(* CODESYS project fserror_0.2.0.1.library
   Company: FisoThemes
   DefaultNamespace: FsError
   Version: 0.2.0.1
   Placeholder: FsError
   Author: Goodwill Mzumala
   Description: A library that offers a set of functions for raising, handling, logging and querying error.
   Title: FsError

Project tree, tasks and I/O mapping:
  libraries: SysFile, * (System); SysTime, 3.5.9.0 (System); SysTypes2 Interfaces, * (System); Tc2_Standard, * (Beckhoff Automation GmbH); Tc2_System, * (Beckhoff Automation GmbH); Tc3_Module, * (Beckhoff Automation GmbH)
  DUTs/
    data type E_AdsReturnCode
    data type E_CodesysCmpError
    data type E_GeneralErrorCode
    data type T_DiskLoggerPath
    data type T_Error
    data type T_ErrorCode
    data type T_ErrorMessage
  GVLs/
    global variables GVL_ErrorDescriptors
  ITFs/
    interface I_Error: Code, Descriptor, IsNotRaised, IsRaised, LogMessage, Message, Timestamp
    interface I_ErrorDescriptor: GetDescription
    interface I_ErrorLogger: Invoke
    interface I_ErrorTimestamp: AsDateTime, GetDate, GetTimeOfDay, Raw
    interface I_MutableError: CopyFrom, RaiseError, SetDescriptor, SetTimestamp
  PARAMs/
    global variables PARAM_Constants
  POUs/
    Error Descriptors/
      function block FB_AdsReturnCodesDescriptor [ST]: GetDescription
      function block FB_CodesysCmpErrorDescriptor [ST]: GetDescription
      function block FB_GeneralCodesDescriptor [ST]: GetDescription
    Errors/
      function F_CreateError [ST]
      function F_CreateErrorFromStartRange [ST]
      function block FB_Error [ST]: Code, Descriptor, IsNotRaised, IsRaised, LogMessage, Message, Timestamp
      function block FB_MutableError [ST]: CopyFrom, RaiseError, SetDescriptor, SetTimestamp
    Loggers/
      function block FB_AdsErrorLogger [ST]: Invoke, SetMessageType
      function block FB_DiskErrorLogger [ST]: CreateLogEntry, AutoFlush, Close, Delimiter, FB_exit, FB_init, Flush, Invoke, IsOpen, LineEnding, Open, SetDelimiter, SetLineEnding, SetTextQualifier, TextQualifier
    Timestamp/
      function block FB_ErrorTimestamp [ST]: AsDateTime, GetDate, GetTimeOfDay, Raw
    program PLAYGROUND [ST]
  Project Information/
    function F_GetCompany [ST]
    function F_GetTitle [ST]
    function F_GetVersion [ST]
  UML/
    Error Class Diagram
    Error Descriptor Class Diagram
    Error Logger Class Diagram
    Error Timestamp Class Diagram
  Version/
    global variables Global_Version
*)

// DUTs/E_AdsReturnCode
// All ADS error codes.
// Source: https://github.com/Roald87/TcError/blob/main/TcError/TcError/ADS/AdsErrorCodes.TcDUT
// See end for licensing information.
{attribute 'qualified_only'}
{attribute 'to_string'}
TYPE E_AdsReturnCode :
(
    ERR_NOERROR 					:= 0,					// No error.
    ERR_INTERNAL,  											// Internal error.
    ERR_NORTIME,  											// No real-time.
    ERR_ALLOCLOCKEDMEM,  									// Allocation locked – memory error.
    ERR_INSERTMAILBOX,  									// Mailbox full – the ADS message could not be sent. Reducing the number of ADS messages per cycle will help.
    ERR_WRONGRECEIVEHMSG,  									// Wrong HMSG.
    ERR_TARGETPORTNOTFOUND,  								// Target port not found – ADS server is not started or is not reachable.
    ERR_TARGETMACHINENOTFOUND,  							// Target computer not found – AMS route was not found.
    ERR_UNKNOWNCMDID, 										// Unknown command ID.
    ERR_BADTASKID,  										// Invalid task ID.
    ERR_NOIO,  												// No IO.
	ERR_UNKNOWNAMSCMD,  									// Unknown AMS command.
    ERR_WIN32ERROR,  										// Win32 error.
    ERR_PORTNOTCONNECTED,  									// Port not connected.
    ERR_INVALIDAMSLENGTH,  									// Invalid AMS length.
    ERR_INVALIDAMSNETID,  									// Invalid AMS Net ID.
    ERR_LOWINSTLEVEL,  										// Installation level is too low –TwinCAT 2 license error.
    ERR_NODEBUGINTAVAILABLE,  								// No debugging available.
    ERR_PORTDISABLED,  										// Port disabled – TwinCAT system service not started.
    ERR_PORTALREADYCONNECTED,  								// Port already connected.
	ERR_AMSSYNC_W32ERROR,  									// AMS Sync Win32 error.
	ERR_AMSSYNC_TIMEOUT,  									// AMS Sync Timeout.
    ERR_AMSSYNC_AMSERROR,  									// AMS Sync error.
    ERR_AMSSYNC_NOINDEXINMAP,  								// No index map for AMS Sync available.
    ERR_INVALIDAMSPORT,  									// Invalid AMS port.
    ERR_NOMEMORY,  											// No memory.
    ERR_TCPSEND,  											// TCP send error.
    ERR_HOSTUNREACHABLE,  									// Host unreachable.
    ERR_INVALIDAMSFRAGMENT,  								// Invalid AMS fragment.
    ERR_TLSSEND,  											// TLS send error – secure ADS connection failed.
    ERR_ACCESSDENIED,  										// Access denied – secure ADS access denied.
    ROUTERERR_NOLOCKEDMEMORY 				:= 1280,		// Locked memory cannot be allocated.
    ROUTERERR_RESIZEMEMORY,  								// The router memory size could not be changed.
	ROUTERERR_MAILBOXFULL,  								// The mailbox has reached the maximum number of possible messages.
    ROUTERERR_DEBUGBOXFULL,  								// The Debug mailbox has reached the maximum number of possible messages.
    ROUTERERR_UNKNOWNPORTTYPE,  							// The port type is unknown.
    ROUTERERR_NOTINITIALIZED,  								// The router is not initialized.
    ROUTERERR_PORTALREADYINUSE,  							// The port number is already assigned.
    ROUTERERR_NOTREGISTERED,  								// The port is not registered.
    ROUTERERR_NOMOREQUEUES,  								// The maximum number of ports has been reached.
    ROUTERERR_INVALIDPORT,  								// The port is invalid.
    ROUTERERR_NOTACTIVATED,  								// The router is not active.
    ROUTERERR_FRAGMENTBOXFULL,  							// The mailbox has reached the maximum number for fragmented messages.
    ROUTERERR_FRAGMENTTIMEOUT,  							// A fragment timeout has occurred.
	ROUTERERR_TOBEREMOVED,  								// The port is removed.
    ADSERR_DEVICE_ERROR 					:= 1792,  		// General device error.
    ADSERR_DEVICE_SRVNOTSUPP,  								// Service is not supported by the server.
    ADSERR_DEVICE_INVALIDGRP,  								// Invalid index group.
    ADSERR_DEVICE_INVALIDOFFSET,  							// Invalid index offset.
    ADSERR_DEVICE_INVALIDACCESS,  							// Reading or writing not permitted.
    ADSERR_DEVICE_INVALIDSIZE,  							// Parameter size not correct.
    ADSERR_DEVICE_INVALIDDATA,  							// Invalid data values.
    ADSERR_DEVICE_NOTREADY,  								// Device is not ready to operate.
    ADSERR_DEVICE_BUSY,  									// Device is busy.
    ADSERR_DEVICE_INVALIDCONTEXT,  							// Invalid operating system context. This can result from use of ADS function blocks in different tasks. It may be possible to resolve this through Multi-task data access synchronization in the PLC.
    ADSERR_DEVICE_NOMEMORY,  								// Insufficient memory.
    ADSERR_DEVICE_INVALIDPARM,  							// Invalid parameter values.
    ADSERR_DEVICE_NOTFOUND,  								// Not found (files, ...).
	ADSERR_DEVICE_SYNTAX,  									// Syntax error in file or command.
    ADSERR_DEVICE_INCOMPATIBLE,  							// Objects do not match.
    ADSERR_DEVICE_EXISTS,  									// Object already exists.
    ADSERR_DEVICE_SYMBOLNOTFOUND,  							// Symbol not found.
    ADSERR_DEVICE_SYMBOLVERSIONINVALID,  					// Invalid symbol version. This can occur due to an online change. Create a new handle.
    ADSERR_DEVICE_INVALIDSTATE,  							// Device (server) is in invalid state.
    ADSERR_DEVICE_TRANSMODENOTSUPP,  						// AdsTransMode not supported.
    ADSERR_DEVICE_NOTIFYHNDINVALID,  						// Notification handle is invalid.
    ADSERR_DEVICE_CLIENTUNKNOWN,  							// Notification client not registered.
    ADSERR_DEVICE_NOMOREHDLS,  								// No further handle available.
    ADSERR_DEVICE_INVALIDWATCHSIZE,  						// Notification size too large.
    ADSERR_DEVICE_NOTINIT,  								// Device not initialized.
    ADSERR_DEVICE_TIMEOUT,  								// Device has a timeout.
    ADSERR_DEVICE_NOINTERFACE,  							// Interface query failed.
    ADSERR_DEVICE_INVALIDINTERFACE,  						// Wrong interface requested.
    ADSERR_DEVICE_INVALIDCLSID,  							// Class ID is invalid.
    ADSERR_DEVICE_INVALIDOBJID,  							// Object ID is invalid.
    ADSERR_DEVICE_PENDING,  								// Request pending.
    ADSERR_DEVICE_ABORTED,  								// Request is aborted.
    ADSERR_DEVICE_WARNING,  								// Signal warning.
    ADSERR_DEVICE_INVALIDARRAYIDX,  						// Invalid array index.
    ADSERR_DEVICE_SYMBOLNOTACTIVE,  						// Symbol not active.
    ADSERR_DEVICE_ACCESSDENIED,  							// Access denied.
    ADSERR_DEVICE_LICENSENOTFOUND,  						// Missing license.
    ADSERR_DEVICE_LICENSEEXPIRED,  							// License expired.
    ADSERR_DEVICE_LICENSEEXCEEDED,  						// License exceeded.
    ADSERR_DEVICE_LICENSEINVALID,  							// Invalid license.
    ADSERR_DEVICE_LICENSESYSTEMID,  						// License problem: System ID is invalid.
    ADSERR_DEVICE_LICENSENOTIMELIMIT,  						// License not limited in time.
    ADSERR_DEVICE_LICENSEFUTUREISSUE,  						// License problem: Time in the future.
    ADSERR_DEVICE_LICENSETIMETOLONG,  						// License period too long.
    ADSERR_DEVICE_EXCEPTION,  								// Exception at system startup.
	ADSERR_DEVICE_LICENSEDUPLICATED,  						// License file read twice.
	ADSERR_DEVICE_SIGNATUREINVALID, 						// License file read twice.
	ADSERR_DEVICE_CERTIFICATEINVALID,  						// Invalid certificate.
    ADSERR_DEVICE_LICENSEOEMNOTFOUND,  						// Public key not known from OEM.
    ADSERR_DEVICE_LICENSERESTRICTED,  						// License not valid for this system ID.
    ADSERR_DEVICE_LICENSEDEMODENIED,  						// Demo license prohibited.
    ADSERR_DEVICE_INVALIDFNCID,  							// Invalid function ID.
    ADSERR_DEVICE_OUTOFRANGE,  								// Outside the valid range.
    ADSERR_DEVICE_INVALIDALIGNMENT,  						// Invalid alignment.
    ADSERR_DEVICE_LICENSEPLATFORM,  						// Invalid platform level.
    ADSERR_DEVICE_FORWARD_PL,  								// Context – forward to passive level.
    ADSERR_DEVICE_FORWARD_DL,  								// Context – forward to dispatch level.
    ADSERR_DEVICE_FORWARD_RT,  								// Context – forward to real-time.
    ADSERR_CLIENT_ERROR 					:= 1856,  		// Client error.
    ADSERR_CLIENT_INVALIDPARM,  							// Service contains an invalid parameter.
    ADSERR_CLIENT_LISTEMPTY,  								// Polling list is empty.
    ADSERR_CLIENT_VARUSED,  								// Var connection already in use.
    ADSERR_CLIENT_DUPLINVOKEID,  							// The called ID is already in use.
    ADSERR_CLIENT_SYNCTIMEOUT,  							// Timeout has occurred – the remote terminal is not responding in the specified ADS timeout. The route setting of the remote terminal may be configured incorrectly.
    ADSERR_CLIENT_W32ERROR,  								// Error in Win32 subsystem.
    ADSERR_CLIENT_TIMEOUTINVALID,  							// Invalid client timeout value.
    ADSERR_CLIENT_PORTNOTOPEN,  							// Port not open.
    ADSERR_CLIENT_NOAMSADDR,  								// No AMS address.
    ADSERR_CLIENT_SYNCINTERNAL,  							// Internal error in Ads sync.
	ADSERR_CLIENT_ADDHASH,  								// Hash table overflow.
    ADSERR_CLIENT_REMOVEHASH,  								// Key not found in the table.
    ADSERR_CLIENT_NOMORESYM,  								// No symbols in the cache.
    ADSERR_CLIENT_SYNCRESINVALID,  							// Invalid response received.
    ADSERR_CLIENT_SYNCPORTLOCKED,  							// Sync Port is locked.
    RTERR_INTERNAL 							:= 4096,  		// Internal error in the real-time system.
    RTERR_BADTIMERPERIODS,  								// Timer value is not valid.
    RTERR_INVALIDTASKPTR,  									// Task pointer has the invalid value 0 (zero).
    RTERR_INVALIDSTACKPTR,  								// Stack pointer has the invalid value 0 (zero).
    RTERR_PRIOEXISTS,  										// The request task priority is already assigned.
    RTERR_NOMORETCB,  										// No free TCB (Task Control Block) available. The maximum number of TCBs is 64.
    RTERR_NOMORESEMAS,  									// No free semaphores available. The maximum number of semaphores is 64.
    RTERR_NOMOREQUEUES,  									// No free space available in the queue. The maximum number of positions in the queue is 64.
    RTERR_EXTIRQALREADYDEF					:= 4109,  		// An external synchronization interrupt is already applied.
    RTERR_EXTIRQNOTDEF,  									// No external sync interrupt applied.
    RTERR_EXTIRQINSTALLFAILED,  							// Application of the external synchronization interrupt has failed.
    RTERR_IRQLNOTLESSOREQUAL,  								// Call of a service function in the wrong context
    RTERR_VMXNOTSUPPORTED					:= 4119,  		// Intel VT-x extension is not supported.
    RTERR_VMXDISABLED,  									// Intel VT-x extension is not enabled in the BIOS.
    RTERR_VMXCONTROLSMISSING,  								// Missing function in Intel VT-x extension.
    RTERR_VMXENABLEFAILS,  									// Activation of Intel VT-x fails.
	WSAETIMEDOUT							:= 10060,		// A connection timeout has occurred while establishing the connection. Either the remote terminal did not respond properly after a certain period of time, or the established connection could not be maintained because the connected host did not respond.
    WSAECONNREFUSED							:= 10061,		// Connection refused. Connection couldn't be established because the target computer has rejected it. Error can result from an attempt to connect to a service that is inactive on the external host, i.e. a service for which no server application is running.
    WSAEHOSTUNREACH							:= 10065,		// No route to host - a socket operation referred to an unavailable host.
	ERR_UNKNOWN                       		:= 4294967294	// Unknown ADS error code.
)LINT;
END_TYPE
(*
	MIT License
	
	Copyright (c) 2022 Roald87
	
	Permission is hereby granted, free of charge, to any person obtaining a copy
	of this software and associated documentation files (the "Software"), to deal
	in the Software without restriction, including without limitation the rights
	to use, copy, modify, merge, publish, distribute, sublicense, and/or sell
	copies of the Software, and to permit persons to whom the Software is
	furnished to do so, subject to the following conditions:
	
	The above copyright notice and this permission notice shall be included in all
	copies or substantial portions of the Software.
	
	THE SOFTWARE IS PROVIDED "AS IS", WITHOUT WARRANTY OF ANY KIND, EXPRESS OR
	IMPLIED, INCLUDING BUT NOT LIMITED TO THE WARRANTIES OF MERCHANTABILITY,
	FITNESS FOR A PARTICULAR PURPOSE AND NONINFRINGEMENT. IN NO EVENT SHALL THE
	AUTHORS OR COPYRIGHT HOLDERS BE LIABLE FOR ANY CLAIM, DAMAGES OR OTHER
	LIABILITY, WHETHER IN AN ACTION OF CONTRACT, TORT OR OTHERWISE, ARISING FROM,
	OUT OF OR IN CONNECTION WITH THE SOFTWARE OR THE USE OR OTHER DEALINGS IN THE
	SOFTWARE.
*)

// DUTs/E_CodesysCmpError
 // Error codes are found @ CmpErrors.Errors.<variable> from the CmpErrors2 Interfaces library.
 // See: https://help.codesys.com/webapp/Errors;product=CmpErrors2_Itfs;version=3.5.15.0
{attribute 'qualified_only'}
{attribute 'to_string'}
TYPE E_CodesysCmpError :
(
	ERR_OK 						 := 16#0,	//	Ok
	ERR_FAILED 					 := 16#1, 	//	General error - To be used only for internal errors
	ERR_PARAMETER 				 := 16#2, 	//	Invalid parameter for this operation
	ERR_NOT_INITIALIZED 		 := 16#3, 	//	Function cannot be executed, since component has not been initialized yet. It may work later, though
	ERR_VERSION 				 := 16#4, 	//	Version conflict
	ERR_TIMEOUT 				 := 16#5, 	//	Operation timed out
	ERR_NO_BUFFER 				 := 16#6, 	//	Insufficient memory to carry out the request
	ERR_PENDING 				 := 16#A, 	//	For async-calls: call not complete, yet
	ERR_NUM_PENDING 			 := 16#B, 	//  Too many pending calls. Try later
	ERR_NOT_IMPLEMENTED 		 := 16#C, 	//  The function is not implemented
	ERR_INVALID_ID 				 := 16#D, 	//  No object with the provided id found
	ERR_OVERFLOW 				 := 16#E, 	//	Integer overflow
	ERR_BUFFER_SIZE 			 := 16#F, 	//	The size of a buffer is too small OR invalid
	ERR_NO_OBJECT 				 := 16#10,	//	No object with this specified name available
	ERR_NO_MEMORY 				 := 16#11,	//  No heap memory available
	ERR_DUPLICATE 				 := 16#12, 	//  An object with the same name is still available
	ERR_MEMORY_OVERWRITE 		 := 16#13,  //  Heap memory was written out of bounds! Memory overwrite error
	ERR_INVALID_HANDLE 			 := 16#14,  //  Invalid handle to an object
	ERR_END_OF_0BJECT 			 := 16#15,  //  End OF object reached
	ERR_NO_CHANGE 				 := 16#16,  //  No changes done
	ERR_INVALID_INTERFACE 		 := 16#17,  //  Invalid or unknown interface
	ERR_NOT_SUPPORTED 			 := 16#18,  //  Functionality not supported
	ERR_NO_ACCESS_RIGHTS 		 := 16#19,  //  No access rights for this operation
	ERR_OUT_OF_LIMITS 			 := 16#1A,  //  Specified limits of a resource exceeded
	ERR_ENTRIES_REMAINING 		 := 16#1B,  //  Remaining entries that could not be transmitted because of buffer limitation
	ERR_INVALID_SESSION_ID 		 := 16#1C,  //  Invalid online sessionid
	ERR_EXCEPTION 				 := 16#1D,  //  Exception occurred
	ERR_SIGNATURE_MISMATCH 		 := 16#1E,	//	Signature mismatch of an api function
	ERR_VERSION_MISMATCH 		 := 16#1F,	//	Version mismatch
	ERR_TYPE_MISMATCH 			 := 16#20,	//	Type mismatch
	ERR_ID_MISMATCH 			 := 16#21,	//	ID mismatch
	ERR_NO_CONSISTENCY 			 := 16#22,	//	Consistency error
	ERR_NO_COMM_CYCLE 			 := 16#23,	//	No COMM_CYCLE needed
	ERR_DONT_SUSPEND_TASK 		 := 16#24,	//	Do not suspend task after an exception
	ERR_MEMORY_LOCK_FAILED 		 := 16#25,	//	Memory cannot be locked in this operation
	ERR_LICENSE_MISSING 		 := 16#26,	//	License missing for the runtime
	ERR_OPERATION_DENIED 		 := 16#27,	//	Operation denied 
	ERR_DEVICE 					 := 16#28,	//	Device error
	ERR_DISK_FULL 				 := 16#29,	//	Disk full
	ERR_CRC_FAILED 				 := 16#30,	//	Internal use in runtime
	ERR_MEDIA_ERASE 			 := 16#31,	//	Internal use in runtime
	ERR_FILE_ERROR 				 := 16#32,	//	File error. e.g. cannot open a file for writing because it could be write protected
	ERR_NO_RETAIN_MEMORY 		 := 16#33,	//	No retain memory available
	ERR_OUT_OF_LIMITS_MIN 		 := 16#34,	//	Specified minimum-limit of a resource exceeded
	ERR_OUT_OF_LIMITS_MAX 		 := 16#35,	//	Specified maximum-limit of a resource exceeded
	ERR_SIZE_MISMATCH 			 := 16#36,	//	Size mismatch
	ERR_CALL_AGAIN 				 := 16#37,	//	Operation is not yet finished, call function again to proceed
	ERR_NOTHING_TO_DO 			 := 16#38,	//	Operation has nothing to do. No execution.
	ERR_SECURITY_CHECKS_FAILED 	 := 16#39,	//	Some security checks have failed. /* This is a generic error code to report this error over public channels. In this case the error code doesn’t provide a detailed cause for the error. */
	ERR_INVALID_SEQUENCE 		 := 16#3A,	//	 
	ERR_INVALID_REFERENCE 		 := 16#3B,	//	Dereferencing an IEC reference in IecVarAccess failed due to invalid destination address, e. G. NULL.
	ERR_CONVERSION_INCOMPLETE 	 := 16#3C,	//	Conversion of string encodings was not lossless.
	ERR_SOCK_NOT_INITIALIZED 	 := 16#201, //  Socket errors (range: 0x0200 - 0X02FF)
	ERR_SOCK_NOT_SOCKET 		 := 16#202, //  The provided socket handle is invalid
	ERR_SOCK_AF_UNSUPPORTED 	 := 16#203, //  The address family is not supported
	ERR_SOCK_PROTO_UNSUPPORTED   := 16#204, //  Protocol is not supported 
	ERR_SOCK_NO_BUFFER 			 := 16#205, //  Not enough buffer to handle the request 
	ERR_SOCK_WOULD_BLOCK 		 := 167206, //  Socket is in nonblocking mode but this call would block 
	ERR_SOCK_ADDR_INUSE 		 := 16#207, //  The provided address is already in use 
	ERR_SOCK_ADDR_NOT_AVAILABLE  := 16#208, //  The provided address is not available on THIS computer 
	ERR_SOCK_CONN_REFUSED 		 := 16#209, //  Connection has been refused by the remote host 
	ERR_SOCK_TIMEDOUT 			 := 16#20A, //  Operation timed out
	ERR_SOCK_HOST_NOT_FOUND 	 := 16#20B, //  The host has NOT been found
	ERR_SOCK_HOST_UNREACHABLE  	 := 16#20C, //  Host is unreachable
	ERR_SOCK_1S_CONNECTED 		 := 16#20D, //  Socket is already connected
	ERR_SOCK_NOT_CONNECTED 		 := 16#20E, //  The socket is not connected
	ERR_SOCK_SHUTDOWN 			 := 16#20F, //  Shutdown has been called on the socket 
	ERR_SOCK_MSGSIZE 			 := 16#210, //  For sockets of type DGRAM. The package to send exceeds the maximum package size 
	ERR_SOCK_CLOSED 			 := 16#211, //  Socket has been gracefully closed. No more send/receives allowed 
	ERR_L7_TAG_MISSING 			 := 16#300,	//  Tag missing in online communication buffer
	ERR_L7_UNKNOWN_CMD_GROUP 	 := 16#301,	//  Unknown command group
	ERR_L7_UNKNOWN_CMD 			 := 16#302,	//  Unknown command (within a valid command group)
	ERR_L7_INCOMPLETE 			 := 16#303	//  Level 7 service incomplete
)LINT;
END_TYPE

// DUTs/E_GeneralErrorCode
// List of general error codes used in a system.
{attribute 'qualified_only'}
{attribute 'to_string'}
TYPE E_GeneralErrorCode :
(
	{region "General Errors (1-99)"}
	ERR_NO_ERROR                    := 0,      // No error.
	ERR_GENERAL_ERROR               := 1,      // General error - To be used only for internal errors
	ERR_INVALID_PARAMETER           := 2,      // Invalid parameter for this operation
	ERR_NOT_INITIALIZED             := 3,      // Function cannot be executed since the component has not been initialized yet. It may work later, though
	ERR_VERSION_CONFLICT            := 4,      // Version conflict
	{endregion}
	
	{region "Overflow Errors (100-119)"}
	ERR_INTEGER_OVERFLOW            := 100,    // Integer overflow
	ERR_BUFFER_OVERFLOW             := 101,    // Buffer overflow
	ERR_STACK_OVERFLOW              := 102,    // Stack overflow
	ERR_HEAP_OVERFLOW               := 103,    // Heap overflow
	{endregion}
	
	{region "Buffer Errors (120-139)"}
	ERR_NO_BUFFER                   := 120,    // No buffer available
	ERR_BUFFER_UNDERFLOW            := 121,    // Buffer underflow
	ERR_BUFFER_FULL                 := 123,    // Buffer is full
	{endregion}
	
	{region "Configuration and Settings Errors (140-159)"}
	ERR_INVALID_CONFIGURATION       := 140,    // Invalid configuration or settings
	ERR_CONFIGURATION_MISSING       := 141,    // Required configuration setting or parameter is missing
	{endregion}
	
	{region "Network Errors (200-249)"}
	ERR_NETWORK_ERROR               := 200,    // Network communication or connectivity issues
	ERR_TIMEOUT_CONNECT             := 201,    // Connection timeout
	ERR_TIMEOUT_READ                := 202,    // Read timeout
	ERR_TIMEOUT_WRITE               := 203,    // Write timeout
	ERR_UNSUPPORTED_FORMAT          := 204,    // Unsupported data format
	ERR_TOO_MANY_REQUESTS           := 205,    // Too many requests or actions in a short period
	{endregion}
	
	{region "Stream Errors (250-299)"}
	ERR_STREAM_ERROR                := 250,    // Generic stream error
	ERR_STREAM_NOT_FOUND            := 251,    // Stream not found
	ERR_STREAM_READ_FAILED          := 252,    // Stream read operation failed
	ERR_STREAM_WRITE_FAILED         := 253,    // Stream write operation failed
	ERR_STREAM_PERMISSION_DENIED    := 254,    // Stream operation permission denied
	ERR_STREAM_ALREADY_EXISTS       := 255,    // Stream already exists
	{endregion}
	
	{region "Resource Errors (300-339)"}
	ERR_NOT_FOUND                   := 300,    // The resource has not been found
	ERR_PERMISSION_DENIED           := 301,    // Permission denied
	ERR_DATA_NOT_AVAILABLE          := 302,    // Requested data is not available
	ERR_OUT_OF_BOUNDS               := 303,    // Value is outside the valid range
	ERR_DATA_CORRUPTED              := 304,    // Data corruption or integrity issues
	ERR_INVALID_INTERFACE           := 305,    // Invalid or unknown interface
	ERR_INVALID_REFERENCE           := 306,    // Dereferencing an IEC reference in IecVarAccess failed due to an invalid destination address, e.g., NULL.
	ERR_INVALID_POINTER             := 307,    // Invalid pointer
	ERR_INVALID_HANDLE              := 308,    // Invalid handle to an object
	ERR_MIN_LIMIT_EXCEEDED          := 309,    // Specified minimum-limit of the resource exceeded
	ERR_MAX_LIMIT_EXCEEDED          := 310,    // Specified maximum-limit of the resource exceeded
	ERR_DUPLICATE                   := 311,    // The resource already exists
	{endregion}
	
	{region "Hardware Errors (400-449)"}
	ERR_HARDWARE_FAILURE            := 400,    // Hardware malfunctions or failures
	{endregion}
	
	{region "Resource Management Errors (500-549)"}
	ERR_RESOURCE_BUSY               := 500,    // Resource is currently in use and cannot be accessed
	ERR_RESOURCE_LOCKED             := 501,    // Resource is locked and cannot be accessed
	{endregion}
	
	{region "State and Operation Errors (600-649)"}
	ERR_INVALID_STATE               := 600,    // Invalid state for the requested operation
	ERR_INVALID_OPERATION           := 601,    // Requested operation is not allowed or valid in the current context
	ERR_OPERATION_TIMEOUT           := 602,    // Operation timed out
	ERR_OPERATION_FAILED            := 603,    // Operation failed
	{endregion}
	
	{region "Service and API Errors (700-749)"}
	ERR_EXTERNAL_SERVICE_FAILURE    := 700,    // Failure in an external service or API
	ERR_UNAVAILABLE_SERVICE         := 701,    // Required service or component is not available
	{endregion}
	
	{region "Data Conversion Errors (800-849)"}
	ERR_INVALID_INPUT               := 800,   // Invalid or unexpected input provided
	ERR_INVALID_CONVERSION          := 801,   // Invalid data conversion
	ERR_INVALID_COMPARISON          := 802,   // Invalid comparison
	ERR_TYPE_MISMATCH               := 803,   // Type mismatch
	ERR_SIZE_MISMATCH               := 804,   // Size mismatch
	{endregion}
	
	{region "Security Errors (900-949)"}
	ERR_SECURITY_CHECKS_FAILED      := 900,   // Some security checks have failed. (Generic error for reporting over public channels)
	ERR_AUTHENTICATION_FAILED       := 901,   // Authentication process failed
	ERR_AUTHORIZATION_FAILED        := 902,   // Authorization failed due to insufficient permissions
	{endregion}
	
	{region "Memory Errors (1000-1049)"}
	ERR_MEMORY_ALLOCATION_FAILED    := 1000,  // Memory allocation failed
	ERR_INSUFFICIENT_MEMORY         := 1001,  // Insufficient memory to carry out the request
	ERR_INSUFFICIENT_MEMORY_FULL    := 1002,  // Memory full
	{endregion}
	
	{region "File Errors (1100-1149)"}
	ERR_FILE_NOT_FOUND              := 1100,  // The specified file was not found
	ERR_FILE_READ_FAILED            := 1101,  // File read operation failed
	ERR_FILE_WRITE_FAILED           := 1102,  // File write operation failed
	ERR_FILE_PERMISSION_DENIED      := 1103,  // File operation permission denied
	ERR_FILE_ALREADY_EXISTS         := 1104,  // File already exists
	ERR_FILE_TOO_LARGE              := 1105,  // File size exceeds the maximum allowed size
	ERR_FILE_FORMAT_UNSUPPORTED     := 1106,  // Unsupported file format
	ERR_FILE_NOT_OPEN				:= 1107,  // File isn't open
	ERR_FILE_INVALID_HANDLE			:= 1108,  // File handle is invalid
	{endregion}
	
	{region "Directory Errors (1150-1199)"}
	ERR_DIRECTORY_NOT_FOUND         := 1150,  // The specified directory was not found
	ERR_DIRECTORY_READ_FAILED       := 1151,  // Directory read operation failed
	ERR_DIRECTORY_WRITE_FAILED      := 1152,  // Directory write operation failed
	ERR_DIRECTORY_PERMISSION_DENIED := 1153,  // Directory operation permission denied
	ERR_DIRECTORY_NOT_EMPTY         := 1154,  // Directory is not empty
	ERR_DIRECTORY_ALREADY_EXISTS    := 1155,  // Directory already exists
	ERR_DIRECTORY_NOT_OPEN			:= 1157,  // Directory isn't open
	ERR_DIRECTORY_INVALID_HANDLE	:= 1158,  // Directory handle is invalid
	{endregion}
	
	{region "Cache Errors (1200-1249)"}
	ERR_CACHE_MISS                  := 1200,  // Cache miss occurred
	ERR_CACHE_WRITE_FAILED          := 1201,  // Cache write operation failed
	{endregion}
	
	{region "Serialization/Deserialization Errors (1300-1349)"}
	ERR_SERIALIZATION_FAILED        := 1300,  // Data serialization failed
	ERR_DESERIALIZATION_FAILED      := 1301,  // Data deserialization failed
	{endregion}
	
	{region "Threading and Concurrency Errors (1400-1449)"}
	ERR_THREAD_CREATION_FAILED      := 1400,  // Thread creation failed
	ERR_DEADLOCK_DETECTED           := 1401,  // Deadlock detected
	ERR_CONCURRENCY_VIOLATION       := 1402,  // Concurrency violation
	{endregion}
	
	{region "Protocol Errors (1500-1549)"}
	ERR_PROTOCOL_VIOLATION          := 1500,  // Protocol violation detected
	ERR_UNSUPPORTED_PROTOCOL        := 1501,  // Unsupported protocol
	{endregion}
	
	{region "User Errors (1600-1699)"}
	ERR_USER_INPUT_INVALID          := 1600,  // User input is invalid or malformed
	ERR_USER_INPUT_TOO_LONG         := 1601,  // User input exceeds maximum allowed length
	ERR_USER_INPUT_TOO_SHORT        := 1602,  // User input is shorter than the minimum required length
	ERR_USER_AUTHENTICATION_FAILED  := 1603,  // User authentication failed
	ERR_USER_AUTHORIZATION_FAILED   := 1604,  // User is not authorized to perform this action
	ERR_USER_ACCOUNT_LOCKED         := 1605,  // User account is locked
	ERR_USER_ACCOUNT_DISABLED       := 1606,  // User account is disabled
	ERR_USER_SESSION_EXPIRED        := 1607,  // User session has expired
	ERR_USER_ALREADY_EXISTS         := 1608,  // User already exists
	ERR_USER_NOT_FOUND              := 1609,  // User not found
	ERR_USER_CANCELLED              := 1610,  // User cancelled the operation or action
	{endregion}
	
	{region "Internal additional errors (5000-5099)"}
	ERR_NOTHING_TO_DO               := 5000,  // Operation has nothing to do. No execution.
	ERR_FUNCTION_NOT_SUPPORTED      := 5001,  // Functionality not supported
	{endregion}
	
	{region "Custom errors (10000-99999)"}
	ERR_CUSTOM_ERROR_BEGIN          := 10_000,  // Custom or application-specific error codes can be defined starting from here
	ERR_CUSTOM_ERROR_END          	:= 99_999,  // Custom or application-specific error codes definition ends here
	{endregion}
	
	{region "Codesys errors (200000-299999)"} 
	ERR_CODESYS_BEGIN				:= 100_000, // Start range of Codesys errors in the context of general errors
	ERR_CODESYS_END					:= 999_999,	// End range of Codesys errors in the context of general errors
	{endregion}
	
	{region "ADS errors (1,000,000,000-...)"} 
	ERR_ADS_RETURN_CODE_BEGIN		:= 1_000_000_000, // Start range of ADS return codes in the context of general errors
	ERR_ADS_RETURN_CODE_END 		:= ERR_ADS_RETURN_CODE_BEGIN + 4_294_967_294 // End range of ADS return codes in the context of general errors
	{endregion}
) LINT;
END_TYPE

// DUTs/T_DiskLoggerPath
TYPE T_DiskLoggerPath : STRING(PARAM_Constants.DISK_LOGGER_PATH_LENGTH); END_TYPE

// DUTs/T_Error
// Alias for the error object.
TYPE T_Error : FB_Error; END_TYPE

// DUTs/T_ErrorCode
// Alias for error code.
TYPE T_ErrorCode : LINT; END_TYPE

// DUTs/T_ErrorMessage
// Alias for error messages as strings with a predefined maximum length.
// Length of message can be changed in the **Library_Parameters**.
TYPE T_ErrorMessage : STRING(PARAM_Constants.ERROR_MESSAGE_SIZE); END_TYPE

// GVLs/GVL_ErrorDescriptors
{attribute 'qualified_only'}
VAR_GLOBAL
	fbAdsReturnCodes	: FB_AdsReturnCodesDescriptor;
	fbCodesysCmpErrors 	: FB_CodesysCmpErrorDescriptor;
	fbGeneralErrorCodes	: FB_GeneralCodesDescriptor;
END_VAR

// PARAMs/PARAM_Constants
// Main parameters for the library.
{attribute 'qualified_only'}
VAR_GLOBAL CONSTANT
	ERROR_MESSAGE_SIZE 				: __UXINT := 255; // String length of an error message.
	DISK_LOGGER_PATH_LENGTH			: __UXINT := 300; // String length of disk logger path.
END_VAR

// Version/Global_Version
{attribute 'TcGenerated'}
{attribute 'no-analysis'}
{attribute 'linkalways'}
// This function has been automatically generated from the project information.
VAR_GLOBAL CONSTANT
	{attribute 'const_non_replaced'}
	stLibVersion_FsError : ST_LibVersion := (iMajor := 0, iMinor := 2, iBuild := 0, iRevision := 1, nFlags := 0, sVersion := '0.2.0.1');
END_VAR

// ITFs/I_Error
// This interface represents an error with a code, message, timestamp, a raised status as well as logging capabilities.
INTERFACE I_Error EXTENDS __SYSTEM.IQueryInterface

// The error code associated with this error.
// [get] Returns the error code.
PROPERTY Code : T_ErrorCode
GET
END_GET
END_PROPERTY

// The provider for error code descriptions.
// [get] Returns the error code descriptor.
PROPERTY Descriptor : I_ErrorDescriptor
GET
END_GET
END_PROPERTY

// A boolean flag indicating whether the error has been raised.
// [get] Returns TRUE if the error has **NOT** been raised, FALSE otherwise.
PROPERTY IsNotRaised : BOOL
GET
END_GET
END_PROPERTY

// A boolean flag indicating whether the error has been raised.
// [get] Returns TRUE if the error has been raised, FALSE otherwise.
PROPERTY IsRaised : BOOL
GET
END_GET
END_PROPERTY

// Logs this error message using the provided logger.
METHOD LogMessage : I_Error // Reference to the current instance of I_Error
VAR_INPUT
	ipLogger 	: I_ErrorLogger; 	// The logger to use for logging.
END_VAR
VAR_OUTPUT
	bIsBusy 	: BOOL;				// Is the operation still executing?
	Error 		: T_Error;			// Error produced by operation.
END_VAR
END_METHOD

// A descriptive message providing more details about the error.
// [get] Returns the error message.
PROPERTY Message : T_ErrorMessage
GET
END_GET
END_PROPERTY

// The timestamp indicating when this error message occurred.
// [get] Returns the timestamp.
PROPERTY Timestamp : I_ErrorTimestamp
GET
END_GET
END_PROPERTY

END_INTERFACE

// ITFs/I_ErrorDescriptor
// This interface provides a method to retrieve descriptive messages for error codes.
INTERFACE I_ErrorDescriptor EXTENDS __SYSTEM.IQueryInterface;

// Retrieves the descriptive message for the specified error code.
METHOD GetDescription : T_ErrorMessage // The descriptive message corresponding to the provided error code.
VAR_INPUT
	Code : T_ErrorCode; // The error code for which the description is to be retrieved.
END_VAR
END_METHOD

END_INTERFACE

// ITFs/I_ErrorLogger
// This interface represents a logger for error messages.
INTERFACE I_ErrorLogger EXTENDS __SYSTEM.IQueryInterface

// Logs the provided error message.
METHOD Invoke
VAR_INPUT
	ipError : I_Error;	 // The error message to be logged.
END_VAR
VAR_OUTPUT
	bIsBusy : BOOL;		// Is the operation still executing?
	Error 	: T_Error;	// Error produced by operation.
END_VAR
END_METHOD

END_INTERFACE

// ITFs/I_ErrorTimestamp
// Interface that represents a timestamp and provides methods to retrieve various date and time components.
INTERFACE I_ErrorTimestamp EXTENDS __SYSTEM.IQueryInterface

// Retrieves the timestamp as a combined date and time value.
METHOD AsDateTime : DT // The combined date and time value as a DT (Date and Time).
VAR_INPUT
END_VAR
END_METHOD

// Retrieves the date part of the timestamp.
METHOD GetDate : DATE // The date part of the timestamp.
VAR_INPUT
END_VAR
END_METHOD

// Retrieves the time of day part of the timestamp.
METHOD GetTimeOfDay : TOD // The time of day part of the timestamp.
VAR_INPUT
END_VAR
END_METHOD

// The raw timestamp value which represents the number of milliseconds since Thursday, 1.1.1970 00:00:00.000.
// [get] Returns the raw timestamp value.
PROPERTY Raw : ULINT
GET
END_GET
END_PROPERTY

END_INTERFACE

// ITFs/I_MutableError
// This interface represents an error that is mutable.
INTERFACE I_MutableError EXTENDS I_Error

// Copies the properties from another error instance.
// This method allows the current mutable error instance to copy the error code,
// descriptor, message, and timestamp from another error instance, effectively
// duplicating the state of the provided error instance.
METHOD CopyFrom : I_MutableError // A reference to the current instance.
VAR_INPUT
	ipError : I_Error; // The error instance from which to copy the properties
END_VAR
END_METHOD

// Raises an error with the specified error code.
METHOD RaiseError : I_MutableError // A reference to the current instance.
VAR_INPUT
    Code : T_ErrorCode; // The error code to raise.
END_VAR
END_METHOD

// Sets the error descriptor
METHOD SetDescriptor : I_MutableError // A reference to the current instance.
VAR_INPUT
    ipDescriptor : I_ErrorDescriptor; // The error descriptor to set.
END_VAR
END_METHOD

// Sets the timestamp of the error.
METHOD SetTimestamp : I_MutableError // A reference to the current instance.
VAR_INPUT
	nTimestamp : ULINT; // High resolution timestamp of when the error occured.
END_VAR
END_METHOD

END_INTERFACE

// POUs/Error Descriptors/FB_AdsReturnCodesDescriptor
// Descriptor for ADS errors codes.
// Provides description for errors.
{attribute 'no_assign'}
{attribute 'enable_dynamic_creation'}
{attribute 'no_explicit_call' := 'direct call for this function block is not allowed'}
FUNCTION_BLOCK FINAL FB_AdsReturnCodesDescriptor IMPLEMENTS I_ErrorDescriptor
VAR
END_VAR

// Retrieves the descriptive message for the specified error code.
METHOD GetDescription : T_ErrorMessage // The descriptive message corresponding to the provided error code.
VAR_INPUT
	Code : T_ErrorCode; // The error code for which the description is to be retrieved.
END_VAR
CASE Code OF
    E_AdsReturnCode.ERR_NOERROR:						GetDescription := 'No error.';
    E_AdsReturnCode.ERR_INTERNAL:						GetDescription := 'Internal error.';
    E_AdsReturnCode.ERR_NORTIME:						GetDescription := 'No real-time.';
    E_AdsReturnCode.ERR_ALLOCLOCKEDMEM:					GetDescription := 'Allocation locked – memory error.';
    E_AdsReturnCode.ERR_INSERTMAILBOX:					GetDescription := 'Mailbox full - the ADS message could not be sent. Reducing the number of ADS messages per cycle will help.';
    E_AdsReturnCode.ERR_WRONGRECEIVEHMSG:				GetDescription := 'Wrong HMSG.';
    E_AdsReturnCode.ERR_TARGETPORTNOTFOUND:				GetDescription := 'Target port not found – ADS server is not started or is not reachable.';
    E_AdsReturnCode.ERR_TARGETMACHINENOTFOUND:			GetDescription := 'Target computer not found – AMS route was not found.';
    E_AdsReturnCode.ERR_UNKNOWNCMDID:					GetDescription := 'Unknown command ID.';
    E_AdsReturnCode.ERR_BADTASKID:						GetDescription := 'Invalid task ID.';
    E_AdsReturnCode.ERR_NOIO:							GetDescription := 'No IO.';
    E_AdsReturnCode.ERR_UNKNOWNAMSCMD:					GetDescription := 'Unknown AMS command.';
    E_AdsReturnCode.ERR_WIN32ERROR:						GetDescription := 'Win32 error.';
    E_AdsReturnCode.ERR_PORTNOTCONNECTED:				GetDescription := 'Port not connected.';
    E_AdsReturnCode.ERR_INVALIDAMSLENGTH:				GetDescription := 'Invalid AMS length.';
    E_AdsReturnCode.ERR_INVALIDAMSNETID:				GetDescription := 'Invalid AMS Net ID.';
    E_AdsReturnCode.ERR_LOWINSTLEVEL:					GetDescription := 'Installation level is too low –TwinCAT 2 license error.';
    E_AdsReturnCode.ERR_NODEBUGINTAVAILABLE:			GetDescription := 'No debugging available.';
    E_AdsReturnCode.ERR_PORTDISABLED:					GetDescription := 'Port disabled – TwinCAT system service not started.';
    E_AdsReturnCode.ERR_PORTALREADYCONNECTED:			GetDescription := 'Port already connected.';
    E_AdsReturnCode.ERR_AMSSYNC_W32ERROR:				GetDescription := 'AMS Sync Win32 error.';
    E_AdsReturnCode.ERR_AMSSYNC_TIMEOUT: 				GetDescription := 'AMS Sync Timeout.';
    E_AdsReturnCode.ERR_AMSSYNC_AMSERROR: 				GetDescription := 'AMS Sync error.';
    E_AdsReturnCode.ERR_AMSSYNC_NOINDEXINMAP: 			GetDescription := 'No index map for AMS Sync available.';
    E_AdsReturnCode.ERR_INVALIDAMSPORT: 				GetDescription := 'Invalid AMS port.';
    E_AdsReturnCode.ERR_NOMEMORY: 						GetDescription := 'No memory.';
    E_AdsReturnCode.ERR_TCPSEND:						GetDescription := 'TCP send error.';
    E_AdsReturnCode.ERR_HOSTUNREACHABLE:				GetDescription := 'Host unreachable.';
    E_AdsReturnCode.ERR_INVALIDAMSFRAGMENT:				GetDescription := 'Invalid AMS fragment.';
    E_AdsReturnCode.ERR_TLSSEND:						GetDescription := 'TLS send error - secure ADS connection failed.';
    E_AdsReturnCode.ERR_ACCESSDENIED:					GetDescription := 'Access denied - secure ADS access denied.';
    E_AdsReturnCode.ROUTERERR_NOLOCKEDMEMORY:			GetDescription := 'Locked memory cannot be allocated.';
    E_AdsReturnCode.ROUTERERR_RESIZEMEMORY:				GetDescription := 'The router memory size could not be changed.';
    E_AdsReturnCode.ROUTERERR_MAILBOXFULL:				GetDescription := 'The mailbox has reached the maximum number of possible messages.';
    E_AdsReturnCode.ROUTERERR_DEBUGBOXFULL:				GetDescription := 'The Debug mailbox has reached the maximum number of possible messages.';
    E_AdsReturnCode.ROUTERERR_UNKNOWNPORTTYPE: 			GetDescription := 'The port type is unknown.';
    E_AdsReturnCode.ROUTERERR_NOTINITIALIZED: 			GetDescription := 'The router is not initialized.';
    E_AdsReturnCode.ROUTERERR_PORTALREADYINUSE: 		GetDescription := 'The port number is already assigned.';
    E_AdsReturnCode.ROUTERERR_NOTREGISTERED: 			GetDescription := 'The port is not registered.';
    E_AdsReturnCode.ROUTERERR_NOMOREQUEUES:				GetDescription := 'The maximum number of ports has been reached.';
    E_AdsReturnCode.ROUTERERR_INVALIDPORT:				GetDescription := 'The port is invalid.';
    E_AdsReturnCode.ROUTERERR_NOTACTIVATED:				GetDescription := 'The router is not active.';
    E_AdsReturnCode.ROUTERERR_FRAGMENTBOXFULL:			GetDescription := 'The mailbox has reached the maximum number for fragmented messages.';
    E_AdsReturnCode.ROUTERERR_FRAGMENTTIMEOUT:			GetDescription := 'A fragment timeout has occurred.';
    E_AdsReturnCode.ROUTERERR_TOBEREMOVED:				GetDescription := 'The port is removed.';
    E_AdsReturnCode.ADSERR_DEVICE_ERROR:				GetDescription := 'General device error.';
    E_AdsReturnCode.ADSERR_DEVICE_SRVNOTSUPP:			GetDescription := 'Service is not supported by the server.';
    E_AdsReturnCode.ADSERR_DEVICE_INVALIDGRP:			GetDescription := 'Invalid index group.';
    E_AdsReturnCode.ADSERR_DEVICE_INVALIDOFFSET:		GetDescription := 'Invalid index offset.';
    E_AdsReturnCode.ADSERR_DEVICE_INVALIDACCESS:		GetDescription := 'Reading or writing not permitted.';
    E_AdsReturnCode.ADSERR_DEVICE_INVALIDSIZE:			GetDescription := 'Parameter size not correct.';
    E_AdsReturnCode.ADSERR_DEVICE_INVALIDDATA:			GetDescription := 'Invalid data values.';
    E_AdsReturnCode.ADSERR_DEVICE_NOTREADY:				GetDescription := 'Device is not ready to operate.';
    E_AdsReturnCode.ADSERR_DEVICE_BUSY:					GetDescription := 'Device is busy.';
    E_AdsReturnCode.ADSERR_DEVICE_INVALIDCONTEXT:		GetDescription := 'Invalid operating system context. This can result from use of ADS function blocks in different tasks. It may be possible to resolve this through Multi-task data access synchronization in the PLC.';
    E_AdsReturnCode.ADSERR_DEVICE_NOMEMORY:				GetDescription := 'Insufficient memory.';
    E_AdsReturnCode.ADSERR_DEVICE_INVALIDPARM:			GetDescription := 'Invalid parameter values.';
    E_AdsReturnCode.ADSERR_DEVICE_NOTFOUND:				GetDescription := 'Not found (files, ...).';
    E_AdsReturnCode.ADSERR_DEVICE_SYNTAX:				GetDescription := 'Syntax error in file or command.';
    E_AdsReturnCode.ADSERR_DEVICE_INCOMPATIBLE:			GetDescription := 'Objects do not match.';
    E_AdsReturnCode.ADSERR_DEVICE_EXISTS:				GetDescription := 'Object already exists.';
    E_AdsReturnCode.ADSERR_DEVICE_SYMBOLNOTFOUND:		GetDescription := 'Symbol not found.';
    E_AdsReturnCode.ADSERR_DEVICE_SYMBOLVERSIONINVALID:	GetDescription := 'Invalid symbol version. This can occur due to an online change. Create a new handle.';
    E_AdsReturnCode.ADSERR_DEVICE_INVALIDSTATE:			GetDescription := 'Device (server) is in invalid state.';
    E_AdsReturnCode.ADSERR_DEVICE_TRANSMODENOTSUPP:		GetDescription := 'AdsTransMode not supported.';
    E_AdsReturnCode.ADSERR_DEVICE_NOTIFYHNDINVALID:		GetDescription := 'Notification handle is invalid.';
    E_AdsReturnCode.ADSERR_DEVICE_CLIENTUNKNOWN:		GetDescription := 'Notification client not registered.';
    E_AdsReturnCode.ADSERR_DEVICE_NOMOREHDLS:			GetDescription := 'No further handle available.';
    E_AdsReturnCode.ADSERR_DEVICE_INVALIDWATCHSIZE:		GetDescription := 'Notification size too large.';
    E_AdsReturnCode.ADSERR_DEVICE_NOTINIT:				GetDescription := 'Device not initialized.';
    E_AdsReturnCode.ADSERR_DEVICE_TIMEOUT:				GetDescription := 'Device has a timeout.';
    E_AdsReturnCode.ADSERR_DEVICE_NOINTERFACE:			GetDescription := 'Interface query failed.';
    E_AdsReturnCode.ADSERR_DEVICE_INVALIDINTERFACE:		GetDescription := 'Wrong interface requested.';
    E_AdsReturnCode.ADSERR_DEVICE_INVALIDCLSID:			GetDescription := 'Class ID is invalid.';
    E_AdsReturnCode.ADSERR_DEVICE_INVALIDOBJID:			GetDescription := 'Object ID is invalid.';
    E_AdsReturnCode.ADSERR_DEVICE_PENDING:				GetDescription := 'Request pending.';
    E_AdsReturnCode.ADSERR_DEVICE_ABORTED:				GetDescription := 'Request is aborted.';
    E_AdsReturnCode.ADSERR_DEVICE_WARNING:				GetDescription := 'Signal warning.';
    E_AdsReturnCode.ADSERR_DEVICE_INVALIDARRAYIDX:		GetDescription := 'Invalid array index.';
    E_AdsReturnCode.ADSERR_DEVICE_SYMBOLNOTACTIVE:		GetDescription := 'Symbol not active.';
    E_AdsReturnCode.ADSERR_DEVICE_ACCESSDENIED:			GetDescription := 'Access denied.';
    E_AdsReturnCode.ADSERR_DEVICE_LICENSENOTFOUND:		GetDescription := 'Missing license.';
    E_AdsReturnCode.ADSERR_DEVICE_LICENSEEXPIRED:		GetDescription := 'License expired.';
    E_AdsReturnCode.ADSERR_DEVICE_LICENSEEXCEEDED:		GetDescription := 'License exceeded.';
    E_AdsReturnCode.ADSERR_DEVICE_LICENSEINVALID:		GetDescription := 'Invalid license.';
    E_AdsReturnCode.ADSERR_DEVICE_LICENSESYSTEMID:		GetDescription := 'License problem: System ID is invalid.';
    E_AdsReturnCode.ADSERR_DEVICE_LICENSENOTIMELIMIT:	GetDescription := 'License not limited in time.';
    E_AdsReturnCode.ADSERR_DEVICE_LICENSEFUTUREISSUE:	GetDescription := 'License problem: Time in the future.';
    E_AdsReturnCode.ADSERR_DEVICE_LICENSETIMETOLONG:	GetDescription := 'License period too long.';
    E_AdsReturnCode.ADSERR_DEVICE_EXCEPTION:			GetDescription := 'Exception at system startup.';
    E_AdsReturnCode.ADSERR_DEVICE_LICENSEDUPLICATED:	GetDescription := 'License file read twice.';
    E_AdsReturnCode.ADSERR_DEVICE_SIGNATUREINVALID:		GetDescription := 'Invalid signature.';
    E_AdsReturnCode.ADSERR_DEVICE_CERTIFICATEINVALID:	GetDescription := 'Invalid certificate.';
    E_AdsReturnCode.ADSERR_DEVICE_LICENSEOEMNOTFOUND:	GetDescription := 'Public key not known from OEM.';
    E_AdsReturnCode.ADSERR_DEVICE_LICENSERESTRICTED:	GetDescription := 'License not valid for this system ID.';
    E_AdsReturnCode.ADSERR_DEVICE_LICENSEDEMODENIED:	GetDescription := 'Demo license prohibited.';
    E_AdsReturnCode.ADSERR_DEVICE_INVALIDFNCID:			GetDescription := 'Invalid function ID.';
    E_AdsReturnCode.ADSERR_DEVICE_OUTOFRANGE:			GetDescription := 'Outside the valid range.';
    E_AdsReturnCode.ADSERR_DEVICE_INVALIDALIGNMENT:		GetDescription := 'Invalid alignment.';
    E_AdsReturnCode.ADSERR_DEVICE_LICENSEPLATFORM:		GetDescription := 'Invalid platform level.';
    E_AdsReturnCode.ADSERR_DEVICE_FORWARD_PL:			GetDescription := 'Context – forward to passive level.';
    E_AdsReturnCode.ADSERR_DEVICE_FORWARD_DL:			GetDescription := 'Context – forward to dispatch level.';
    E_AdsReturnCode.ADSERR_DEVICE_FORWARD_RT:			GetDescription := 'Context – forward to real-time.';
    E_AdsReturnCode.ADSERR_CLIENT_ERROR:				GetDescription := 'Client error.';
    E_AdsReturnCode.ADSERR_CLIENT_INVALIDPARM:			GetDescription := 'Service contains an invalid parameter.';
    E_AdsReturnCode.ADSERR_CLIENT_LISTEMPTY:			GetDescription := 'Polling list is empty.';
    E_AdsReturnCode.ADSERR_CLIENT_VARUSED:				GetDescription := 'Var connection already in use.';
    E_AdsReturnCode.ADSERR_CLIENT_DUPLINVOKEID:			GetDescription := 'The called ID is already in use.';
    E_AdsReturnCode.ADSERR_CLIENT_SYNCTIMEOUT:			GetDescription := 'Timeout has occurred - the remote terminal is not responding in the specified ADS timeout. The route setting of the remote terminal may be configured incorrectly.';
    E_AdsReturnCode.ADSERR_CLIENT_W32ERROR:				GetDescription := 'Error in Win32 subsystem.';
    E_AdsReturnCode.ADSERR_CLIENT_TIMEOUTINVALID:		GetDescription := 'Invalid client timeout value.';
    E_AdsReturnCode.ADSERR_CLIENT_PORTNOTOPEN:			GetDescription := 'Port not open.';
    E_AdsReturnCode.ADSERR_CLIENT_NOAMSADDR:			GetDescription := 'No AMS address.';
    E_AdsReturnCode.ADSERR_CLIENT_SYNCINTERNAL:			GetDescription := 'Internal error in Ads sync.';
    E_AdsReturnCode.ADSERR_CLIENT_ADDHASH:				GetDescription := 'Hash table overflow.';
    E_AdsReturnCode.ADSERR_CLIENT_REMOVEHASH:			GetDescription := 'Key not found in the table.';
    E_AdsReturnCode.ADSERR_CLIENT_NOMORESYM:			GetDescription := 'No symbols in the cache.';
    E_AdsReturnCode.ADSERR_CLIENT_SYNCRESINVALID:		GetDescription := 'Invalid response received.';
    E_AdsReturnCode.ADSERR_CLIENT_SYNCPORTLOCKED:		GetDescription := 'Sync Port is locked.';
    E_AdsReturnCode.RTERR_INTERNAL:						GetDescription := 'Internal error in the real-time system.';
    E_AdsReturnCode.RTERR_BADTIMERPERIODS:				GetDescription := 'Timer value is not valid.';
    E_AdsReturnCode.RTERR_INVALIDTASKPTR:				GetDescription := 'Task pointer has the invalid value 0 (zero).';
    E_AdsReturnCode.RTERR_INVALIDSTACKPTR:				GetDescription := 'Stack pointer has the invalid value 0 (zero).';
    E_AdsReturnCode.RTERR_PRIOEXISTS:					GetDescription := 'The request task priority is already assigned.';
    E_AdsReturnCode.RTERR_NOMORETCB:					GetDescription := 'No free TCB (Task Control Block) available. The maximum number of TCBs is 64.';
    E_AdsReturnCode.RTERR_NOMORESEMAS:					GetDescription := 'No free semaphores available. The maximum number of semaphores is 64.';
    E_AdsReturnCode.RTERR_NOMOREQUEUES:					GetDescription := 'No free space available in the queue. The maximum number of positions in the queue is 64.';
    E_AdsReturnCode.RTERR_EXTIRQALREADYDEF:				GetDescription := 'An external synchronization interrupt is already applied.';
    E_AdsReturnCode.RTERR_EXTIRQNOTDEF:					GetDescription := 'No external sync interrupt applied.';
    E_AdsReturnCode.RTERR_EXTIRQINSTALLFAILED:			GetDescription := 'Application of the external synchronization interrupt has failed.';
    E_AdsReturnCode.RTERR_IRQLNOTLESSOREQUAL:			GetDescription := 'Call of a service function in the wrong context';
    E_AdsReturnCode.RTERR_VMXNOTSUPPORTED:				GetDescription := 'Intel VT-x extension is not supported.';
    E_AdsReturnCode.RTERR_VMXDISABLED:					GetDescription := 'Intel VT-x extension is not enabled in the BIOS.';
    E_AdsReturnCode.RTERR_VMXCONTROLSMISSING:			GetDescription := 'Missing function in Intel VT-x extension.';
    E_AdsReturnCode.RTERR_VMXENABLEFAILS:				GetDescription := 'Activation of Intel VT-x fails.';
    E_AdsReturnCode.WSAETIMEDOUT: 						GetDescription := 'A connection timeout has occurred while establishing the connection. Either the remote terminal did not respond properly after a certain period of time, or the established connection could not be maintained because the connected host did not respond.';
    E_AdsReturnCode.WSAECONNREFUSED: 					GetDescription := 'Connection refused. Connection couldnt be established because the target computer has rejected it. Error can result from an attempt to connect to a service that is inactive on the external host, i.e. a service for which no server application is running.';
    E_AdsReturnCode.WSAEHOSTUNREACH: 					GetDescription := 'No route to host - a socket operation referred to an unavailable host.';
ELSE
    GetDescription := Tc2_Standard.CONCAT('Unknown ADS error code: ', Tc2_Standard.CONCAT(TO_STRING(Code), '.'));
	END_CASE
END_METHOD

END_FUNCTION_BLOCK

// POUs/Error Descriptors/FB_CodesysCmpErrorDescriptor
// Descriptor for Codesys CmpErrors.
// Provides description for errors.
{attribute 'no_assign'}
{attribute 'enable_dynamic_creation'}
{attribute 'no_explicit_call' := 'direct call for this function block is not allowed'}
FUNCTION_BLOCK FB_CodesysCmpErrorDescriptor IMPLEMENTS I_ErrorDescriptor
VAR
END_VAR

// Retrieves the descriptive message for the specified error code.
METHOD GetDescription : T_ErrorMessage // The descriptive message corresponding to the provided error code.
VAR_INPUT
	Code : T_ErrorCode; // The error code for which the description is to be retrieved.
END_VAR
CASE Code OF
    E_CodesysCmpError.ERR_OK:                       GetDescription := 'No error.';
    E_CodesysCmpError.ERR_FAILED:                   GetDescription := 'General error - To be used only for internal errors.';
    E_CodesysCmpError.ERR_PARAMETER:                GetDescription := 'Invalid parameter for this operation.';
    E_CodesysCmpError.ERR_NOT_INITIALIZED:          GetDescription := 'Function cannot be executed, since component has not been initialized yet. It may work later, though.';
    E_CodesysCmpError.ERR_VERSION:                  GetDescription := 'Version conflict.';
    E_CodesysCmpError.ERR_TIMEOUT:                  GetDescription := 'Operation timed out.';
    E_CodesysCmpError.ERR_NO_BUFFER:                GetDescription := 'Insufficient memory to carry out the request.';
    E_CodesysCmpError.ERR_PENDING:                  GetDescription := 'For async-calls: call not complete, yet.';
    E_CodesysCmpError.ERR_NUM_PENDING:              GetDescription := 'Too many pending calls. Try later.';
    E_CodesysCmpError.ERR_NOT_IMPLEMENTED:          GetDescription := 'The function is not implemented.';
    E_CodesysCmpError.ERR_INVALID_ID:               GetDescription := 'No object with the provided id found.';
    E_CodesysCmpError.ERR_OVERFLOW:                 GetDescription := 'Integer overflow.';
    E_CodesysCmpError.ERR_BUFFER_SIZE:              GetDescription := 'The size of a buffer is too small OR invalid.';
    E_CodesysCmpError.ERR_NO_OBJECT:                GetDescription := 'No object with this specified name available.';
    E_CodesysCmpError.ERR_NO_MEMORY:                GetDescription := 'No heap memory available.';
    E_CodesysCmpError.ERR_DUPLICATE:                GetDescription := 'An object with the same name is still available.';
    E_CodesysCmpError.ERR_MEMORY_OVERWRITE:         GetDescription := 'Heap memory was written out of bounds! Memory overwrite error.';
    E_CodesysCmpError.ERR_INVALID_HANDLE:           GetDescription := 'Invalid handle to an object.';
    E_CodesysCmpError.ERR_END_OF_0BJECT:            GetDescription := 'End OF object reached.';
    E_CodesysCmpError.ERR_NO_CHANGE:                GetDescription := 'No changes done.';
    E_CodesysCmpError.ERR_INVALID_INTERFACE:        GetDescription := 'Invalid or unknown interface.';
    E_CodesysCmpError.ERR_NOT_SUPPORTED:            GetDescription := 'Functionality not supported.';
    E_CodesysCmpError.ERR_NO_ACCESS_RIGHTS:         GetDescription := 'No access rights for this operation.';
    E_CodesysCmpError.ERR_OUT_OF_LIMITS:            GetDescription := 'Specified limits of a resource exceeded.';
    E_CodesysCmpError.ERR_ENTRIES_REMAINING:        GetDescription := 'Remaining entries that could not be transmitted because of buffer limitation.';
    E_CodesysCmpError.ERR_INVALID_SESSION_ID:       GetDescription := 'Invalid online sessionid.';
    E_CodesysCmpError.ERR_EXCEPTION:                GetDescription := 'Exception occurred.';
    E_CodesysCmpError.ERR_SIGNATURE_MISMATCH:       GetDescription := 'Signature mismatch of an api function.';
    E_CodesysCmpError.ERR_VERSION_MISMATCH:         GetDescription := 'Version mismatch.';
    E_CodesysCmpError.ERR_TYPE_MISMATCH:            GetDescription := 'Type mismatch.';
    E_CodesysCmpError.ERR_ID_MISMATCH:              GetDescription := 'ID mismatch.';
    E_CodesysCmpError.ERR_NO_CONSISTENCY:           GetDescription := 'Consistency error.';
    E_CodesysCmpError.ERR_NO_COMM_CYCLE:            GetDescription := 'No COMM_CYCLE needed.';
    E_CodesysCmpError.ERR_DONT_SUSPEND_TASK:        GetDescription := 'Do not suspend task after an exception.';
    E_CodesysCmpError.ERR_MEMORY_LOCK_FAILED:       GetDescription := 'Memory cannot be locked in this operation.';
    E_CodesysCmpError.ERR_LICENSE_MISSING:          GetDescription := 'License missing for the runtime.';
    E_CodesysCmpError.ERR_OPERATION_DENIED:         GetDescription := 'Operation denied.';
    E_CodesysCmpError.ERR_DEVICE:                   GetDescription := 'Device error.';
    E_CodesysCmpError.ERR_DISK_FULL:                GetDescription := 'Disk full.';
    E_CodesysCmpError.ERR_CRC_FAILED:               GetDescription := 'Internal use in runtime.';
    E_CodesysCmpError.ERR_MEDIA_ERASE:              GetDescription := 'Internal use in runtime.';
    E_CodesysCmpError.ERR_FILE_ERROR:               GetDescription := 'File error. e.g. cannot open a file for writing because it could be write protected.';
    E_CodesysCmpError.ERR_NO_RETAIN_MEMORY:         GetDescription := 'No retain memory available.';
    E_CodesysCmpError.ERR_OUT_OF_LIMITS_MIN:        GetDescription := 'Specified minimum-limit of a resource exceeded.';
    E_CodesysCmpError.ERR_OUT_OF_LIMITS_MAX:        GetDescription := 'Specified maximum-limit of a resource exceeded.';
    E_CodesysCmpError.ERR_SIZE_MISMATCH:            GetDescription := 'Size mismatch.';
    E_CodesysCmpError.ERR_CALL_AGAIN:               GetDescription := 'Operation is not yet finished, call function again to proceed.';
    E_CodesysCmpError.ERR_NOTHING_TO_DO:            GetDescription := 'Operation has nothing to do. No execution.';
    E_CodesysCmpError.ERR_SECURITY_CHECKS_FAILED:   GetDescription := 'Some security checks have failed.';
    E_CodesysCmpError.ERR_INVALID_SEQUENCE:         GetDescription := 'Invalid sequence of operations.';
    E_CodesysCmpError.ERR_INVALID_REFERENCE:        GetDescription := 'Dereferencing an IEC reference in IecVarAccess failed due to invalid destination address, e. G. NULL.';
    E_CodesysCmpError.ERR_CONVERSION_INCOMPLETE:    GetDescription := 'Conversion of string encodings was not lossless.';
    E_CodesysCmpError.ERR_SOCK_NOT_INITIALIZED:     GetDescription := 'Socket errors (range: 0x0200 - 0X02FF).';
    E_CodesysCmpError.ERR_SOCK_NOT_SOCKET:          GetDescription := 'The provided socket handle is invalid.';
    E_CodesysCmpError.ERR_SOCK_AF_UNSUPPORTED:      GetDescription := 'The address family is not supported.';
    E_CodesysCmpError.ERR_SOCK_PROTO_UNSUPPORTED:   GetDescription := 'Protocol is not supported.';
    E_CodesysCmpError.ERR_SOCK_NO_BUFFER:           GetDescription := 'Not enough buffer to handle the request.';
    E_CodesysCmpError.ERR_SOCK_WOULD_BLOCK:         GetDescription := 'Socket is in nonblocking mode but this call would block.';
    E_CodesysCmpError.ERR_SOCK_ADDR_INUSE:          GetDescription := 'The provided address is already in use.';
    E_CodesysCmpError.ERR_SOCK_ADDR_NOT_AVAILABLE:  GetDescription := 'The provided address is not available on THIS computer.';
    E_CodesysCmpError.ERR_SOCK_CONN_REFUSED:        GetDescription := 'Connection has been refused by the remote host.';
    E_CodesysCmpError.ERR_SOCK_TIMEDOUT:            GetDescription := 'Operation timed out.';
    E_CodesysCmpError.ERR_SOCK_HOST_NOT_FOUND:      GetDescription := 'The host has NOT been found.';
    E_CodesysCmpError.ERR_SOCK_HOST_UNREACHABLE:    GetDescription := 'Host is unreachable.';
    E_CodesysCmpError.ERR_SOCK_1S_CONNECTED:        GetDescription := 'Socket is already connected.';
    E_CodesysCmpError.ERR_SOCK_NOT_CONNECTED:       GetDescription := 'The socket is not connected.';
    E_CodesysCmpError.ERR_SOCK_SHUTDOWN:            GetDescription := 'Shutdown has been called on the socket.';
    E_CodesysCmpError.ERR_SOCK_MSGSIZE:             GetDescription := 'For sockets of type DGRAM. The package to send exceeds the maximum package size.';
    E_CodesysCmpError.ERR_SOCK_CLOSED:              GetDescription := 'Socket has been gracefully closed. No more send/receives allowed.';
    E_CodesysCmpError.ERR_L7_TAG_MISSING:           GetDescription := 'Tag missing in online communication buffer.';
    E_CodesysCmpError.ERR_L7_UNKNOWN_CMD_GROUP:     GetDescription := 'Unknown command group.';
    E_CodesysCmpError.ERR_L7_UNKNOWN_CMD:           GetDescription := 'Unknown command (within a valid command group).';
    E_CodesysCmpError.ERR_L7_INCOMPLETE:            GetDescription := 'Level 7 service incomplete.';
ELSE
    GetDescription := Tc2_Standard.CONCAT('Unknown Codesys Cmp error code: ', Tc2_Standard.CONCAT(TO_STRING(Code), '.'));
	END_CASE;
END_METHOD

END_FUNCTION_BLOCK

// POUs/Error Descriptors/FB_GeneralCodesDescriptor
// Descriptor for ADS errors codes.
// Provides description for errors.
{attribute 'no_assign'}
{attribute 'enable_dynamic_creation'}
{attribute 'no_explicit_call' := 'direct call for this function block is not allowed'}
FUNCTION_BLOCK FINAL FB_GeneralCodesDescriptor IMPLEMENTS I_ErrorDescriptor
VAR
END_VAR

// Retrieves the descriptive message for the specified error code.
METHOD GetDescription : T_ErrorMessage // The descriptive message corresponding to the provided error code.
VAR_INPUT
	Code : T_ErrorCode; // The error code for which the description is to be retrieved.
END_VAR
CASE Code OF
    // No error
    E_GeneralErrorCode.ERR_NO_ERROR:                       GetDescription := 'No error.';

    // General Errors (1-99)
    E_GeneralErrorCode.ERR_GENERAL_ERROR:                   GetDescription := 'General error - To be used only for internal errors.';
    E_GeneralErrorCode.ERR_INVALID_PARAMETER:               GetDescription := 'Invalid parameter for this operation.';
    E_GeneralErrorCode.ERR_NOT_INITIALIZED:                 GetDescription := 'Function cannot be executed since the component has not been initialized yet. It may work later, though.';
    E_GeneralErrorCode.ERR_VERSION_CONFLICT:                GetDescription := 'Version conflict.';

    // Overflow Errors (100-119)
    E_GeneralErrorCode.ERR_INTEGER_OVERFLOW:                GetDescription := 'Integer overflow.';
    E_GeneralErrorCode.ERR_BUFFER_OVERFLOW:                 GetDescription := 'Buffer overflow.';
    E_GeneralErrorCode.ERR_STACK_OVERFLOW:                  GetDescription := 'Stack overflow.';
    E_GeneralErrorCode.ERR_HEAP_OVERFLOW:                   GetDescription := 'Heap overflow.';

    // Buffer Errors (120-139)
    E_GeneralErrorCode.ERR_NO_BUFFER:                       GetDescription := 'No buffer available.';
    E_GeneralErrorCode.ERR_BUFFER_UNDERFLOW:                GetDescription := 'Buffer underflow.';
    E_GeneralErrorCode.ERR_BUFFER_FULL:                     GetDescription := 'Buffer is full.';

    // Configuration and Settings Errors (140-159)
    E_GeneralErrorCode.ERR_INVALID_CONFIGURATION:           GetDescription := 'Invalid configuration or settings.';
    E_GeneralErrorCode.ERR_CONFIGURATION_MISSING:           GetDescription := 'Required configuration setting or parameter is missing.';

    // Network Errors (200-249)
    E_GeneralErrorCode.ERR_NETWORK_ERROR:                   GetDescription := 'Network communication or connectivity issues.';
    E_GeneralErrorCode.ERR_TIMEOUT_CONNECT:                 GetDescription := 'Connection timeout.';
    E_GeneralErrorCode.ERR_TIMEOUT_READ:                    GetDescription := 'Read timeout.';
    E_GeneralErrorCode.ERR_TIMEOUT_WRITE:                   GetDescription := 'Write timeout.';
    E_GeneralErrorCode.ERR_UNSUPPORTED_FORMAT:              GetDescription := 'Unsupported data format.';
    E_GeneralErrorCode.ERR_TOO_MANY_REQUESTS:               GetDescription := 'Too many requests or actions in a short period.';

    // Stream Errors (250-299)
    E_GeneralErrorCode.ERR_STREAM_ERROR:                    GetDescription := 'Generic stream error.';
    E_GeneralErrorCode.ERR_STREAM_NOT_FOUND:                GetDescription := 'Stream not found.';
    E_GeneralErrorCode.ERR_STREAM_READ_FAILED:              GetDescription := 'Stream read operation failed.';
    E_GeneralErrorCode.ERR_STREAM_WRITE_FAILED:             GetDescription := 'Stream write operation failed.';
    E_GeneralErrorCode.ERR_STREAM_PERMISSION_DENIED:        GetDescription := 'Stream operation permission denied.';
    E_GeneralErrorCode.ERR_STREAM_ALREADY_EXISTS:           GetDescription := 'Stream already exists.';

    // Resource Errors (300-339)
    E_GeneralErrorCode.ERR_NOT_FOUND:                       GetDescription := 'The resource has not been found.';
    E_GeneralErrorCode.ERR_PERMISSION_DENIED:               GetDescription := 'Permission denied.';
    E_GeneralErrorCode.ERR_DATA_NOT_AVAILABLE:              GetDescription := 'Requested data is not available.';
    E_GeneralErrorCode.ERR_OUT_OF_BOUNDS:                   GetDescription := 'Value is outside the valid range.';
    E_GeneralErrorCode.ERR_DATA_CORRUPTED:                  GetDescription := 'Data corruption or integrity issues.';
    E_GeneralErrorCode.ERR_INVALID_INTERFACE:               GetDescription := 'Invalid or unknown interface.';
    E_GeneralErrorCode.ERR_INVALID_REFERENCE:               GetDescription := 'Dereferencing an IEC reference in IecVarAccess failed due to an invalid destination address, e.g., NULL.';
    E_GeneralErrorCode.ERR_INVALID_POINTER:                 GetDescription := 'Invalid pointer.';
    E_GeneralErrorCode.ERR_INVALID_HANDLE:                  GetDescription := 'Invalid handle to an object.';
    E_GeneralErrorCode.ERR_MIN_LIMIT_EXCEEDED:              GetDescription := 'Specified minimum-limit of the resource exceeded.';
    E_GeneralErrorCode.ERR_MAX_LIMIT_EXCEEDED:              GetDescription := 'Specified maximum-limit of the resource exceeded.';
    E_GeneralErrorCode.ERR_DUPLICATE:                       GetDescription := 'The resource already exists.';

    // Hardware Errors (400-449)
    E_GeneralErrorCode.ERR_HARDWARE_FAILURE:                GetDescription := 'Hardware malfunctions or failures.';

    // Resource Management Errors (500-549)
    E_GeneralErrorCode.ERR_RESOURCE_BUSY:                   GetDescription := 'Resource is currently in use and cannot be accessed.';
    E_GeneralErrorCode.ERR_RESOURCE_LOCKED:                 GetDescription := 'Resource is locked and cannot be accessed.';

    // State and Operation Errors (600-649)
    E_GeneralErrorCode.ERR_INVALID_STATE:                   GetDescription := 'Invalid state for the requested operation.';
    E_GeneralErrorCode.ERR_INVALID_OPERATION:               GetDescription := 'Requested operation is not allowed or valid in the current context.';
    E_GeneralErrorCode.ERR_OPERATION_TIMEOUT:               GetDescription := 'Operation timed out.';
    E_GeneralErrorCode.ERR_OPERATION_FAILED:                GetDescription := 'Operation failed.';

    // Service and API Errors (700-749)
    E_GeneralErrorCode.ERR_EXTERNAL_SERVICE_FAILURE:        GetDescription := 'Failure in an external service or API';
    E_GeneralErrorCode.ERR_UNAVAILABLE_SERVICE:             GetDescription := 'Required service or component is not available';

    // Data Conversion Errors (800-849)
    E_GeneralErrorCode.ERR_INVALID_INPUT:                   GetDescription := 'Invalid or unexpected input provided.';
    E_GeneralErrorCode.ERR_INVALID_CONVERSION:              GetDescription := 'Invalid data conversion.';
    E_GeneralErrorCode.ERR_INVALID_COMPARISON:              GetDescription := 'Invalid comparison.';
    E_GeneralErrorCode.ERR_TYPE_MISMATCH:                   GetDescription := 'Type mismatch.';
    E_GeneralErrorCode.ERR_SIZE_MISMATCH:                   GetDescription := 'Size mismatch.';

    // Security Errors (900-949)
    E_GeneralErrorCode.ERR_SECURITY_CHECKS_FAILED:          GetDescription := 'Some security checks have failed. (Generic error for reporting over public channels).';
    E_GeneralErrorCode.ERR_AUTHENTICATION_FAILED:           GetDescription := 'Authentication process failed.';
    E_GeneralErrorCode.ERR_AUTHORIZATION_FAILED:            GetDescription := 'Authorization failed due to insufficient permissions.';

    // Memory Errors (1000-1049)
    E_GeneralErrorCode.ERR_MEMORY_ALLOCATION_FAILED:        GetDescription := 'Memory allocation failed.';
    E_GeneralErrorCode.ERR_INSUFFICIENT_MEMORY:             GetDescription := 'Insufficient memory to carry out the request.';
	E_GeneralErrorCode.ERR_INSUFFICIENT_MEMORY_FULL:		GetDescription := 'Memory full.';

    // File Errors (1100-1149)
    E_GeneralErrorCode.ERR_FILE_NOT_FOUND:                  GetDescription := 'The specified file was not found.';
    E_GeneralErrorCode.ERR_FILE_READ_FAILED:                GetDescription := 'File read operation failed.';
    E_GeneralErrorCode.ERR_FILE_WRITE_FAILED:               GetDescription := 'File write operation failed.';
    E_GeneralErrorCode.ERR_FILE_PERMISSION_DENIED:          GetDescription := 'File operation permission denied.';
    E_GeneralErrorCode.ERR_FILE_ALREADY_EXISTS:             GetDescription := 'File already exists.';
    E_GeneralErrorCode.ERR_FILE_TOO_LARGE:                  GetDescription := 'File size exceeds the maximum allowed size.';
    E_GeneralErrorCode.ERR_FILE_FORMAT_UNSUPPORTED:         GetDescription := 'Unsupported file format.';
	E_GeneralErrorCode.ERR_FILE_NOT_OPEN:					GetDescription := 'File isn$'t open.';
	E_GeneralErrorCode.ERR_FILE_INVALID_HANDLE:				GetDescription := 'File handle is invalid.';

    // Directory Errors (1150-1199)
    E_GeneralErrorCode.ERR_DIRECTORY_NOT_FOUND:             GetDescription := 'The specified directory was not found.';
    E_GeneralErrorCode.ERR_DIRECTORY_READ_FAILED:           GetDescription := 'Directory read operation failed.';
    E_GeneralErrorCode.ERR_DIRECTORY_WRITE_FAILED:          GetDescription := 'Directory write operation failed.';
    E_GeneralErrorCode.ERR_DIRECTORY_PERMISSION_DENIED:     GetDescription := 'Directory operation permission denied.';
    E_GeneralErrorCode.ERR_DIRECTORY_NOT_EMPTY:             GetDescription := 'Directory is not empty.';
    E_GeneralErrorCode.ERR_DIRECTORY_ALREADY_EXISTS:        GetDescription := 'Directory already exists.';
	E_GeneralErrorCode.ERR_DIRECTORY_NOT_OPEN:				GetDescription := 'Directory isn$'t open.';
	E_GeneralErrorCode.ERR_DIRECTORY_INVALID_HANDLE:		GetDescription := 'Directory handle is invalid.';

    // Cache Errors (1200-1249)
    E_GeneralErrorCode.ERR_CACHE_MISS:                      GetDescription := 'Cache miss occurred.';
    E_GeneralErrorCode.ERR_CACHE_WRITE_FAILED:              GetDescription := 'Cache write operation failed.';

    // Serialization/Deserialization Errors (1300-1349)
    E_GeneralErrorCode.ERR_SERIALIZATION_FAILED:            GetDescription := 'Data serialization failed.';
    E_GeneralErrorCode.ERR_DESERIALIZATION_FAILED:          GetDescription := 'Data deserialization failed.';

    // Threading and Concurrency Errors (1400-1449)
    E_GeneralErrorCode.ERR_THREAD_CREATION_FAILED:          GetDescription := 'Thread creation failed.';
    E_GeneralErrorCode.ERR_DEADLOCK_DETECTED:               GetDescription := 'Deadlock detected.';
    E_GeneralErrorCode.ERR_CONCURRENCY_VIOLATION:           GetDescription := 'Concurrency violation.';

    // Protocol Errors (1500-1549)
    E_GeneralErrorCode.ERR_PROTOCOL_VIOLATION:              GetDescription := 'Protocol violation detected.';
    E_GeneralErrorCode.ERR_UNSUPPORTED_PROTOCOL:            GetDescription := 'Unsupported protocol.';

    // User Errors (1600-1699)
    E_GeneralErrorCode.ERR_USER_INPUT_INVALID:              GetDescription := 'User input is invalid or malformed.';
    E_GeneralErrorCode.ERR_USER_INPUT_TOO_LONG:             GetDescription := 'User input exceeds maximum allowed length.';
    E_GeneralErrorCode.ERR_USER_INPUT_TOO_SHORT:            GetDescription := 'User input is shorter than the minimum required length.';
    E_GeneralErrorCode.ERR_USER_AUTHENTICATION_FAILED:      GetDescription := 'User authentication failed.';
    E_GeneralErrorCode.ERR_USER_AUTHORIZATION_FAILED:       GetDescription := 'User is not authorized to perform this action.';
	E_GeneralErrorCode.ERR_USER_ACCOUNT_LOCKED:             GetDescription := 'User account is locked.';
    E_GeneralErrorCode.ERR_USER_ACCOUNT_DISABLED:           GetDescription := 'User account is disabled.';
    E_GeneralErrorCode.ERR_USER_SESSION_EXPIRED:            GetDescription := 'User session has expired.';
    E_GeneralErrorCode.ERR_USER_ALREADY_EXISTS:             GetDescription := 'User already exists.';
    E_GeneralErrorCode.ERR_USER_NOT_FOUND:                  GetDescription := 'User not found.';
    E_GeneralErrorCode.ERR_USER_CANCELLED:                  GetDescription := 'User cancelled the operation or action.';

    // Internal additional errors (5000-5099)
    E_GeneralErrorCode.ERR_NOTHING_TO_DO:                   GetDescription := 'Operation has nothing to do. No execution.';
    E_GeneralErrorCode.ERR_FUNCTION_NOT_SUPPORTED:          GetDescription := 'Functionality not supported.';

    // Custom errors (10000-99999)
    E_GeneralErrorCode.ERR_CUSTOM_ERROR_BEGIN
	..E_GeneralErrorCode.ERR_CUSTOM_ERROR_END:              GetDescription := Tc2_Standard.CONCAT(
																				'Custom error code: ',
																				Tc2_Standard.CONCAT(TO_STRING(Code),'.'));
	
	// Codesys errors (10000-99999)
	E_GeneralErrorCode.ERR_CODESYS_BEGIN
	..E_GeneralErrorCode.ERR_CODESYS_END:					GetDescription := Tc2_Standard.CONCAT(
																				'Codesys cmp error code: ', 
																				GVL_ErrorDescriptors
																					.fbCodesysCmpErrors
																					.GetDescription(Code - E_GeneralErrorCode.ERR_CODESYS_BEGIN));
ELSE
    // Because there's a bug with the case state, where it can't read values over 1 million.
	IF Code > E_GeneralErrorCode.ERR_ADS_RETURN_CODE_BEGIN AND Code < E_GeneralErrorCode.ERR_ADS_RETURN_CODE_END THEN
		// ADS errors (1,000,000,000-...)
		GetDescription := Tc2_Standard.CONCAT(
			'ADS return code: ',
			GVL_ErrorDescriptors.fbAdsReturnCodes.GetDescription(Code - E_GeneralErrorCode.ERR_ADS_RETURN_CODE_BEGIN));
	ELSE
		GetDescription := Tc2_Standard.CONCAT('Unknown general error code: ', Tc2_Standard.CONCAT(TO_STRING(Code), '.'));
		END_IF
	END_CASE
END_METHOD

END_FUNCTION_BLOCK

// POUs/Errors/F_CreateError
// Create errors with specified parameters and sets the timestamp to the local time.
FUNCTION F_CreateError : T_Error // Instance of created error.
VAR_INPUT
	ipDescriptor 	: I_ErrorDescriptor; 	// Error descriptor.
	Code 			: T_ErrorCode; 			// Error code.
END_VAR
VAR
	fbMutError 			: FB_MutableError;
	nResult,
	nLowResTimestamp 	: DWORD;
	nHighResTimestamp 	: ULINT;
END_VAR

// Get high res. local timestamp.
nResult := SysTimeRtc.SysTimeRtcConvertUtcToLocal(
			SysTimeRtc.SysTimeRtcGet(nResult),
			nLowResTimestamp);

// Add milliseconds to high res. timestamp.
nHighResTimestamp := TO_ULINT(nLowResTimestamp)*1000 
					 + 
					 (TO_ULINT(LTIME()) MOD TO_ULINT(LTIME#1S)) / TO_ULINT(LTIME#1MS);

// Set muttable error.
fbMutError.SetDescriptor(ipDescriptor)
		  .RaiseError(Code)
		  .SetTimestamp(nHighResTimestamp);
		  
// Return as immutable error.
F_CreateError := fbMutError;

END_FUNCTION

// POUs/Errors/FB_MutableError
// Mutable error object. Used to set error object parameters.
{attribute 'enable_dynamic_creation'}
{attribute 'no_explicit_call' := 'direct call for this function block is not allowed'}
FUNCTION_BLOCK FINAL FB_MutableError EXTENDS FB_Error IMPLEMENTS I_MutableError
VAR
END_VAR

// Copies the properties from another error instance.
// This method allows the current mutable error instance to copy the error code,
// descriptor, message, and timestamp from another error instance, effectively
// duplicating the state of the provided error instance.
METHOD CopyFrom : I_MutableError // A reference to the current instance.
VAR_INPUT
	ipError : I_Error; // The error instance from which to copy the properties
END_VAR
CopyFrom := THIS^;

IF ipError = 0 THEN RETURN; END_IF

THIS^._ipDescriptor := ipError.Descriptor;
THIS^._Code 		:= ipError.Code;
THIS^._nTimestamp	:= ipError.Timestamp.Raw;
END_METHOD

// Raises an error with the specified error code.
METHOD RaiseError  : I_MutableError // A reference to the current instance.
VAR_INPUT
    Code : T_ErrorCode; // The error code to raise.
END_VAR
RaiseError := THIS^;

THIS^._Code := Code;
END_METHOD

// Sets the error descriptor
METHOD SetDescriptor : I_MutableError // A reference to the current instance.
VAR_INPUT
    ipDescriptor : I_ErrorDescriptor; // The error descriptor to set.
END_VAR
SetDescriptor := THIS^;

THIS^._ipDescriptor := ipDescriptor;
END_METHOD

// Sets the timestamp of the error.
METHOD SetTimestamp : I_MutableError // A reference to the current instance.
VAR_INPUT
	nTimestamp : ULINT; // High resolution timestamp of when the error occured.
END_VAR
SetTimestamp := THIS^;

THIS^._nTimestamp := nTimestamp;
END_METHOD

END_FUNCTION_BLOCK

// POUs/Errors/FB_Error
// Base error object. Used to evaluate if an operation as errored out.
{attribute 'enable_dynamic_creation'}
{attribute 'no_explicit_call' := 'direct call for this function block is not allowed'}
FUNCTION_BLOCK FB_Error IMPLEMENTS I_Error
VAR
	_Code 			: T_ErrorCode;
	_nTimestamp		: ULINT;
	_ipDescriptor 	: I_ErrorDescriptor;
END_VAR

// The error code associated with this error.
// [get] Returns the error code.
PROPERTY FINAL Code : T_ErrorCode
GET
Code := THIS^._Code;
END_GET
END_PROPERTY

// The provider for error code descriptions.
// [get] Returns the error code descriptor.
PROPERTY FINAL Descriptor : I_ErrorDescriptor
GET
Descriptor := THIS^._ipDescriptor;
END_GET
END_PROPERTY

// A boolean flag indicating whether the error has been raised.
// [get] Returns TRUE if the error has **NOT** been raised, FALSE otherwise.
PROPERTY IsNotRaised : BOOL
GET
IsNotRaised := NOT THIS^.IsRaised;
END_GET
END_PROPERTY

// A boolean flag indicating whether the error has been raised.
// [get] Returns TRUE if the error has been raised, FALSE otherwise.
PROPERTY FINAL IsRaised : BOOL
GET
IsRaised := THIS^._Code <> 0;
END_GET
END_PROPERTY

// Logs this error message using the provided logger.
METHOD FINAL LogMessage : I_Error // Reference to the current instance of I_Error
VAR_INPUT
	ipLogger 	: I_ErrorLogger; 	// The logger to use for logging.
END_VAR
VAR_OUTPUT
	bIsBusy 	: BOOL;				// Is the operation still executing?
	Error 		: T_Error;			// Error produced by operation.
END_VAR
LogMessage := THIS^;

// Check if interface is valid, if not then return error.
IF ipLogger = 0 THEN 
	Error := F_CreateError(
		GVL_ErrorDescriptors.fbGeneralErrorCodes,
		E_GeneralErrorCode.ERR_INVALID_INTERFACE);
	RETURN;
	END_IF
	
// Invokes the logger.
ipLogger.Invoke(THIS^, bIsBusy => bIsBusy, Error => Error);
END_METHOD

// A descriptive message providing more details about the error.
// [get] Returns the error message.
PROPERTY FINAL Message : T_ErrorMessage
GET
Message := SEL(	THIS^._ipDescriptor <> 0,
				SEL(THIS^._Code = 0, 
					Tc2_Standard.CONCAT('Error raised with code: ', TO_STRING(THIS^.Code)),
					'No Error.'),
				THIS^._ipDescriptor.GetDescription(THIS^.Code));
END_GET
END_PROPERTY

// The timestamp indicating when this error message occurred.
// [get] Returns the timestamp as a DT.
// [warning] Do not assign or call as reference, this is because the
//			 value will be popped off the stack after the first access 
//			 invalidating any references.
PROPERTY Timestamp : I_ErrorTimestamp
GET
VAR_STAT
	fbTimestamp : FB_ErrorTimestamp;
END_VAR
fbTimestamp.Raw := THIS^._nTimestamp;
Timestamp 		:= fbTimestamp;
END_GET
END_PROPERTY

END_FUNCTION_BLOCK

// POUs/Errors/F_CreateErrorFromStartRange
// Create errors with specified parameters and sets the timestamp to the local time from a starting range.
// Some error descriptors have ranges for error codes.
// If the code is 0 an unraised error is created.
FUNCTION F_CreateErrorFromStartRange : T_Error // Instance of created error.
VAR_INPUT
	ipDescriptor 	: I_ErrorDescriptor; 	// Error descriptor.
	StartRange		: T_ErrorCode;			// Error code starting Range. 
	Code 			: T_ErrorCode; 			// Error code.
END_VAR
VAR
	fbMutError 			: FB_MutableError;
	nResult,
	nLowResTimestamp 	: DWORD;
	nHighResTimestamp 	: ULINT;
END_VAR

// Get high res. local timestamp.
nResult := SysTimeRtc.SysTimeRtcConvertUtcToLocal(
			SysTimeRtc.SysTimeRtcGet(nResult),
			nLowResTimestamp);

// Add milliseconds to high res. timestamp.
nHighResTimestamp := TO_ULINT(nLowResTimestamp)*1000 
					 + 
					 (TO_ULINT(LTIME()) MOD TO_ULINT(LTIME#1S)) / TO_ULINT(LTIME#1MS);

// Set muttable error.
fbMutError.SetDescriptor(ipDescriptor)
		  .RaiseError(SEL(Code <> 0, 0, StartRange + Code))
		  .SetTimestamp(nHighResTimestamp);
		  
// Return as immutable error.
F_CreateErrorFromStartRange := fbMutError;

END_FUNCTION

// POUs/Loggers/FB_AdsErrorLogger
// Logs error to ADS logger.
{attribute 'enable_dynamic_creation'}
{attribute 'no_explicit_call' := 'direct call for this function block is not allowed'}
FUNCTION_BLOCK FB_AdsErrorLogger IMPLEMENTS I_ErrorLogger
VAR
	_nMessageType : DWORD := Tc2_System.ADSLOG_MSGTYPE_ERROR;
END_VAR

// Logs the provided error message.
METHOD Invoke
VAR_INPUT
	ipError : I_Error;	 // The error message to be logged.
END_VAR
VAR_OUTPUT
	bIsBusy : BOOL;		// Is the operation still executing?
	Error 	: T_Error;	// Error produced by operation.
END_VAR
VAR
	eResult 			: E_AdsReturnCode;
	sDate, sTimeOfDay 	: STRING(24);
	pDate, pTimeOfDay 	: POINTER TO STRING; 
END_VAR
IF ipError = 0 THEN
	Error := F_CreateError(
		GVL_ErrorDescriptors.fbGeneralErrorCodes,
		E_GeneralErrorCode.ERR_INVALID_INTERFACE);
	RETURN;
	END_IF

sDate 		:= TO_STRING(ipError.Timestamp.GetDate());
sTimeOfDay 	:= TO_STRING(ipError.Timestamp.GetTimeOfDay());

pDate := ADR(sDate[2]);
pTimeOfDay := ADR(sTimeOfDay[4]);


eResult := Tc2_System.ADSLOGSTR(
	THIS^._nMessageType,
	Tc2_Standard.CONCAT(
			Tc2_Standard.CONCAT('Timestamp.: ', Tc2_Standard.CONCAT(pDate^, CONCAT(' ', pTimeOfDay^))), 
			Tc2_Standard.CONCAT(' | Error Code.: %s | Message.: ', ipError.Message)),
	TO_STRING(ipError.Code));

IF eResult <> 0 THEN 
	Error := F_CreateErrorFromStartRange(
		GVL_ErrorDescriptors.fbGeneralErrorCodes,
		E_GeneralErrorCode.ERR_ADS_RETURN_CODE_BEGIN,
		eResult);
	END_IF
END_METHOD

// Determines how the messages should be logged.
// A list of all the control masks for message output currently implemented as global constants in the Tc2_System library.
// See description of the function ADSLOGDINT on infosys under the Tc2_System section.
METHOD SetMessageType : I_ErrorLogger // Reference to the current instance of I_ErrorLogger
VAR_INPUT
	nMessageType : DWORD := Tc2_System.ADSLOG_MSGTYPE_ERROR; // Control mask which determines the type and effect of the message output
END_VAR
SetMessageType := THIS^;

THIS^._nMessageType := nMessageType;
END_METHOD

END_FUNCTION_BLOCK

// POUs/Loggers/FB_DiskErrorLogger
// Simple logger for logging errors to specified file path on disk.
{attribute 'no_assign'}
{attribute 'enable_dynamic_creation'}
{attribute 'no_explicit_call' := 'direct call for this function block is not allowed'}
FUNCTION_BLOCK FB_DiskErrorLogger IMPLEMENTS I_ErrorLogger
VAR
	_FilePath 		: T_DiskLoggerPath;
	_Handle 		: SysTypes.RTS_IEC_HANDLE 	:= SysTypes.RTS_INVALID_HANDLE;
	_bAutoFlush		: BOOL 						:= TRUE;
	_sDelimiter 	: STRING(1) 				:= ',';
	_sTextQualifier : STRING(1) 				:= '"';
	_sLineEnding 	: STRING(10) 				:= '$R$N';
END_VAR

// Creates log entry.
METHOD PROTECTED CreateLogEntry : __XWORD // Size of message.
VAR_IN_OUT
	LoggedErrorMessage 	: T_ErrorMessage; // String to store message.
END_VAR
VAR_INPUT
	ipError				: I_Error;
END_VAR
VAR
	sDate, 
	sTimeOfDay,
	sErrorCode 			: STRING(24);
	ErrorMessage		: T_ErrorMessage;
	nCursor, nIndex 	: __UXINT;
END_VAR
IF ipError = 0 OR SIZEOF(T_ErrorMessage) < 2 THEN RETURN; END_IF

// Convert Date, time of day and error code to string.
sDate 		:= TO_STRING(ipError.Timestamp.GetDate());
sTimeOfDay 	:= TO_STRING(ipError.Timestamp.GetTimeOfDay());
sErrorCode	:= TO_STRING(ipError.Code);

// Append timestamp start text qualifier.
LoggedErrorMessage := THIS^._sTextQualifier;

// Append date.
nIndex := 0;
WHILE sDate[2 + nIndex] <> 0 DO
	nCursor := nCursor + 1;
	LoggedErrorMessage[MIN(nCursor, SIZEOF(T_ErrorMessage))] := sDate[2 + nIndex];
	nIndex := nIndex + 1;
	END_WHILE

// Append space bar.
nCursor := nCursor + 1;
LoggedErrorMessage[MIN(nCursor, SIZEOF(T_ErrorMessage))] := 32;

// Append time of day.
nIndex := 0;
WHILE sTimeOfDay[4 + nIndex] <> 0 DO
	nCursor := nCursor + 1;
	LoggedErrorMessage[MIN(nCursor, SIZEOF(T_ErrorMessage))] := sTimeOfDay[4 + nIndex];
	nIndex := nIndex + 1;
	END_WHILE
	
// Append timestamp end text qualifier.
nCursor := nCursor + 1;
LoggedErrorMessage[MIN(nCursor, SIZEOF(T_ErrorMessage))] := THIS^._sTextQualifier[0];

// Append delimiter.
nCursor := nCursor + 1;
LoggedErrorMessage[MIN(nCursor, SIZEOF(T_ErrorMessage))] := THIS^._sDelimiter[0];

// Append error code start text qualifier.
nCursor := nCursor + 1;
LoggedErrorMessage[MIN(nCursor, SIZEOF(T_ErrorMessage))] := THIS^._sTextQualifier[0];

// Append error code.
nIndex := 0;
WHILE sErrorCode[nIndex] <> 0 DO
	nCursor := nCursor + 1;
	LoggedErrorMessage[MIN(nCursor, SIZEOF(T_ErrorMessage))] := sErrorCode[nIndex];
	nIndex := nIndex + 1;
	END_WHILE
	
// Append error code end text qualifier.
nCursor := nCursor + 1;
LoggedErrorMessage[MIN(nCursor, SIZEOF(T_ErrorMessage))] := THIS^._sTextQualifier[0];

// Append delimiter.
nCursor := nCursor + 1;
LoggedErrorMessage[MIN(nCursor, SIZEOF(T_ErrorMessage))] := THIS^._sDelimiter[0];

// Append error code start text qualifier.
nCursor := nCursor + 1;
LoggedErrorMessage[MIN(nCursor, SIZEOF(T_ErrorMessage))] := THIS^._sTextQualifier[0];

// Append error message.
ErrorMessage := ipError.Message;
nIndex := 0;
WHILE ErrorMessage[nIndex] <> 0 DO
	nCursor := nCursor + 1;
	LoggedErrorMessage[MIN(nCursor, SIZEOF(T_ErrorMessage))] := ErrorMessage[nIndex];
	nIndex := nIndex + 1;
	END_WHILE

// Append error code end text qualifier.
nCursor := nCursor + 1;
LoggedErrorMessage[MIN(nCursor, SIZEOF(T_ErrorMessage))] := THIS^._sTextQualifier[0];

// Append line ending.
nIndex := 0;
WHILE THIS^._sLineEnding[nIndex] <> 0 DO
	nCursor := nCursor + 1;
	LoggedErrorMessage[MIN(nCursor, SIZEOF(T_ErrorMessage))] := THIS^._sLineEnding[nIndex];
	nIndex := nIndex + 1;
	END_WHILE

// Terminate string.
nCursor := nCursor + 1;
LoggedErrorMessage[MIN(nCursor, SIZEOF(T_ErrorMessage))] := 0;

// Return size of string.
CreateLogEntry := SEL(nCursor <> 0, 0, nCursor - 1);
END_METHOD

// Flush the file cache automatically after logging?
// [default] TRUE - Flush after every write.
// [get] Returns the state of the auto-flush config.
// [set] Set the state of the auto-flush config.
PROPERTY AutoFlush : BOOL
GET
AutoFlush := THIS^._bAutoFlush;
END_GET
SET
THIS^._bAutoFlush := AutoFlush;
END_SET
END_PROPERTY

// Closes current log file.
METHOD Close
VAR_OUTPUT
	bIsBusy 	: BOOL;				// Is the operation still executing?
	Error 		: T_Error;			// Error produced by operation.
END_VAR
VAR
	eResult 	: E_CodesysCmpError;
END_VAR
eResult := SysFile.SysFileClose(THIS^._Handle);

IF eResult = E_CodesysCmpError.ERR_OK THEN RETURN; END_IF

Error := F_CreateErrorFromStartRange(
	GVL_ErrorDescriptors.fbGeneralErrorCodes,
	E_GeneralErrorCode.ERR_CODESYS_BEGIN,
	eResult);
END_METHOD

// The character used to separate logger entry fields.
// [default] ','.
// [get] Returns the delimter.
// [set] Sets the delimiter.
PROPERTY Delimiter : STRING(1)
GET
Delimiter := THIS^._sDelimiter;
END_GET
SET
THIS^._sDelimiter := Delimiter;
END_SET
END_PROPERTY

{attribute 'hide'}
METHOD FB_exit : BOOL
VAR_INPUT
	bInCopyCode : BOOL; // if TRUE, the exit method is called for exiting an instance that is copied afterwards (online change).
END_VAR
THIS^.Close();
END_METHOD

{attribute 'hide'}
METHOD FB_init : BOOL
VAR_INPUT
	bInitRetains 	: BOOL; 	// if TRUE, the retain variables are initialized (warm start / cold start)
	bInCopyCode 	: BOOL;  	// if TRUE, the instance afterwards gets moved into the copy code (online change)
	FilePath		: T_DiskLoggerPath;
END_VAR
THIS^._FilePath := FilePath;
END_METHOD

// Flushes the file cache.
METHOD Flush : I_ErrorLogger // Reference to the current instance of error logger.
VAR_OUTPUT
	bIsBusy 	: BOOL;				// Is the operation still executing?
	Error 		: T_Error;			// Error produced by operation.
END_VAR
VAR
	eResult 	: E_CodesysCmpError;
END_VAR
Flush := THIS^;

IF NOT THIS^.IsOpen THEN 
	Error := F_CreateError(
		GVL_ErrorDescriptors.fbGeneralErrorCodes,
		E_GeneralErrorCode.ERR_FILE_NOT_OPEN);
	RETURN;
	END_IF

eResult := SysFile.SysFileFlush(THIS^._Handle);

IF eResult = E_CodesysCmpError.ERR_OK THEN RETURN; end_if

Error := F_CreateErrorFromStartRange(
	GVL_ErrorDescriptors.fbGeneralErrorCodes,
	E_GeneralErrorCode.ERR_CODESYS_BEGIN,
	eResult);
END_METHOD

// Logs the provided error message.
METHOD Invoke
VAR_INPUT
	ipError : I_Error;	 // The error message to be logged.
END_VAR
VAR_OUTPUT
	bIsBusy : BOOL;		// Is the operation still executing?
	Error 	: T_Error;	// Error produced by operation.
END_VAR
VAR
	LoggedErrorMessage 	: T_MaxString;
	nBytesWritten 		: __XWORD;
	eResult 			: E_CodesysCmpError;
END_VAR
IF ipError = 0 THEN
	Error := F_CreateError(
		GVL_ErrorDescriptors.fbGeneralErrorCodes,
		E_GeneralErrorCode.ERR_INVALID_INTERFACE);
	RETURN;
	END_IF

// Open file if it's not open.
IF NOT THIS^.IsOpen THEN 
	THIS^.Open(bIsBusy => bIsBusy, Error => Error);
	IF Error.IsRaised OR bIsBusy THEN RETURN; END_IF 
	END_IF

// Write to disk.
nBytesWritten := SysFile.SysFileWrite(
	THIS^._Handle, ADR(LoggedErrorMessage),
	THIS^.CreateLogEntry(LoggedErrorMessage, ipError), ADR(eResult));

// Check for errors.
IF eResult <> E_CodesysCmpError.ERR_OK THEN 
	Error := F_CreateErrorFromStartRange(
		GVL_ErrorDescriptors.fbGeneralErrorCodes, 
		E_GeneralErrorCode.ERR_CODESYS_BEGIN, 
		eResult);
	END_IF
	
// Check if writter is busy.
bIsBusy := Error.IsNotRaised AND nBytesWritten = 0;

// Flush if not busy and auto-flush is enabled.
IF NOT bIsBusy AND Error.IsNotRaised AND THIS^._bAutoFlush THEN 
	eResult := SysFile.SysFileFlush(THIS^._Handle);
	IF eResult <> E_CodesysCmpError.ERR_OK THEN 
		Error := F_CreateErrorFromStartRange(
			GVL_ErrorDescriptors.fbGeneralErrorCodes, 
			E_GeneralErrorCode.ERR_CODESYS_BEGIN, 
			eResult);
		END_IF
	END_IF
END_METHOD

// Boolean flag indicating whether log file path is open.
// [get] Returns TRUE if the file has been openned, FALSE otherwise.
PROPERTY IsOpen : BOOL
GET
IsOpen := THIS^._Handle <> SysTypes.RTS_INVALID_HANDLE;
END_GET
END_PROPERTY

// The string used to terminate the error log entry.
// [default] '$R$N'.
// [get] Returns the line-ending.
// [set] Sets the line-ending.
PROPERTY LineEnding : STRING(1)
GET
LineEnding := THIS^._sLineEnding;
END_GET
SET
THIS^._sLineEnding := LineEnding;
END_SET
END_PROPERTY

// Opens logger file, creates it if it doesn't exist.
METHOD Open : I_ErrorLogger // Reference to the current instance of error logger.
VAR_OUTPUT
	bIsBusy 	: BOOL;				// Is the operation still executing?
	Error 		: T_Error;			// Error produced by operation.
END_VAR
VAR
	eResult 	: E_CodesysCmpError;
END_VAR
Open := THIS^;

IF THIS^.IsOpen THEN RETURN; END_IF

THIS^._Handle := SysFile.SysFileOpen(THIS^._FilePath, SysFile.AM_APPEND_PLUS, ADR(eResult));

bIsBusy := eResult = E_CodesysCmpError.ERR_OK AND THIS^._Handle = SysTypes.RTS_INVALID_HANDLE;

IF bIsBusy OR eResult = E_CodesysCmpError.ERR_OK THEN RETURN; END_IF

Error := F_CreateErrorFromStartRange(
	GVL_ErrorDescriptors.fbGeneralErrorCodes,
	E_GeneralErrorCode.ERR_CODESYS_BEGIN,
	eResult);
END_METHOD

// Sets the character used to separate logger entry fields.
// [default] ','
METHOD SetDelimiter : REFERENCE TO FB_DiskErrorLogger // Reference to the current instance of error logger.
VAR_INPUT
	sValue : STRING(1); // Delimiter character.
END_VAR
SetDelimiter REF= THIS^;

THIS^._sDelimiter := sValue;
END_METHOD

// Sets the value of the string used to terminate the error log entry.
// [default] '$R$N'.
METHOD SetLineEnding : REFERENCE TO FB_DiskErrorLogger // Reference to the current instance of error logger.
VAR_INPUT
	sValue : STRING(10); // Line ending characters.
END_VAR
SetLineEnding REF= THIS^;

THIS^._sLineEnding := sValue;
END_METHOD

// Sets the character used to enclose logger entry fields.
// [default] '"'.
METHOD SetTextQualifier : REFERENCE TO FB_DiskErrorLogger // Reference to the current instance of error logger.
VAR_INPUT
	sValue : STRING(1); // Text Qualifier character.
END_VAR
SetTextQualifier REF= THIS^;

THIS^._sTextQualifier := sValue;
END_METHOD

// The character used to enclose logger entry fields.
// [default] '"'.
// [get] Returns the text qualifier.
// [set] Set the text qualifier.
PROPERTY TextQualifier : STRING(1)
GET
TextQualifier := THIS^._sTextQualifier;
END_GET
SET
THIS^._sTextQualifier := TextQualifier;
END_SET
END_PROPERTY

END_FUNCTION_BLOCK

// POUs/Timestamp/FB_ErrorTimestamp
{attribute 'enable_dynamic_creation'}
{attribute 'no_explicit_call' := 'direct call for this function block is not allowed'}
FUNCTION_BLOCK FB_ErrorTimestamp IMPLEMENTS I_ErrorTimestamp
VAR
	_nTimestamp : ULINT;
END_VAR

// Retrieves the timestamp as a combined date and time value.
METHOD AsDateTime : DT // The combined date and time value as a DT (Date and Time).
VAR_INPUT
END_VAR
AsDateTime := TO_DT(THIS^._nTimestamp/1000);
END_METHOD

// Retrieves the date part of the timestamp.
METHOD GetDate : DATE // The date part of the timestamp.
VAR_INPUT
END_VAR
GetDate := TO_DATE(THIS^._nTimestamp/1000);
END_METHOD

// Retrieves the time of day part of the timestamp.
METHOD GetTimeOfDay : TOD // The time of day part of the timestamp.
VAR_INPUT
END_VAR
GetTimeOfDay := TO_TOD(THIS^._nTimestamp MOD 86400000);
END_METHOD

// The raw timestamp value which represents the number of milliseconds since Thursday, 1.1.1970 00:00:00.000.
// [get] Returns the raw timestamp value.
// [set] Sets the raw timestamp value.
PROPERTY Raw : ULINT
GET
Raw := THIS^._nTimestamp;
END_GET
SET
THIS^._nTimestamp := Raw;
END_SET
END_PROPERTY

END_FUNCTION_BLOCK

// POUs/PLAYGROUND
{attribute 'no_explicit_call' := 'direct call for this program is not allowed'} 
PROGRAM INTERNAL PLAYGROUND
VAR
	sDate 			: T_ErrorMessage;
	nTimestamp 		: ULINT;
	nSize 			: LINT;
	bCreate,
	bLog 			: BOOL;
	Err				: T_Error;
	fbWithAdsLogger : FB_AdsErrorLogger;
	fbToDisk		: FB_DiskErrorLogger('C:\temp\errlog.csv');
END_VAR
VAR_TEMP
	DiskLogErr 		: T_Error;
END_VAR

nSize := SIZEOF(Err);

IF bCreate THEN 
	bCreate := FALSE;
	Err := F_CreateError(GVL_ErrorDescriptors.fbGeneralErrorCodes,
						 E_GeneralErrorCode.ERR_ADS_RETURN_CODE_BEGIN + E_AdsReturnCode.ADSERR_DEVICE_INVALIDCONTEXT);
	END_IF

IF bLog THEN Err.LogMessage(fbToDisk, bIsBusy => bLog, Error => DiskLogErr); END_IF
	
IF DiskLogErr.IsRaised THEN DiskLogErr.LogMessage(fbWithAdsLogger); END_IF

END_PROGRAM

// Project Information/F_GetCompany
// This function has been automatically generated from the project information.
{attribute 'signature_flag' := '1073741824'}
{attribute 'TcGenerated'}
{attribute 'no-analysis'}
FUNCTION F_GetCompany : WSTRING
VAR_INPUT
	
END_VAR

F_GetCompany := "FisoThemes";

END_FUNCTION

// Project Information/F_GetTitle
// This function has been automatically generated from the project information.
{attribute 'signature_flag' := '1073741824'}
{attribute 'TcGenerated'}
{attribute 'no-analysis'}
FUNCTION F_GetTitle : WSTRING
VAR_INPUT
	
END_VAR

F_GetTitle := "FsError";

END_FUNCTION

// Project Information/F_GetVersion
// This function has been automatically generated from the project information.
{attribute 'signature_flag' := '1073741824'}
{attribute 'TcGenerated'}
{attribute 'no-analysis'}
FUNCTION F_GetVersion : ST_LibVersion
VAR_INPUT
	
END_VAR

F_GetVersion.iMajor := 0;
F_GetVersion.iMinor := 2;
F_GetVersion.iBuild := 0;
F_GetVersion.iRevision := 1;

END_FUNCTION
